(* CODESYS project BE_Framework BA.project

Project tree, tasks and I/O mapping:
  Device : TxB SoftControl, Beijer Electronics Products AB, version 3.5.1.45
    application AREA1
      Symbols
      Struct/
        Sensors/
          data type strSensor1
          data type strSensor2_Regulator
          data type strSensor3_RegOutsideCompensation
          data type strSensor4_FanGuard
          data type strSensor5_FreezeProtection
          data type strSensor6_HeatExchanger_Rot
          data type strSensor7_Humidity
          data type strSensor8_DefrostProtection
          data type strSensor9_CO2
          data type strSensor10_HeatExchanger_Pressure
          data type strSensor11_DifferentialPressure
        Fans/
          data type strFan_Analog
          data type strFan_TwoSpeed
          data type strFan_Onespeed
        Dampers/
          data type strDamper_Digital
          data type strDamper_Analog
        Pumps/
          data type strPumpExercise
          data type strPump
        Valves/
          data type strValveExercise
          data type strValve
        Functions/
          data type strFunction_OutsideCompensation
          data type strFunction_Overtime
          data type strFunction_NightCooling
          data type strFunction_NightHeating
        System/
          data type strSystemTags
          data type strArrayDateTime
          data type strManMode
          data type strSummerTime
        HeatExchangers/
          data type strHeatExchanger_Rot
          data type strHeatExchanger_Cross
        TimeChannels/
          data type strTCH_1StartStop
          data type strTCH_2StartStop
        Units/
          data type strLB
          data type strUC
        IO_Crevis/
          data type strST2792
          data type strST4491
          data type strST1218
          data type strST3708
      System/
        libraries: Standard, * (System); SysTimeRtc, 3.5.1.0 (System); BE Lib BA, 1.1.0.0 (Beijer Electronics)
        task MainTask (cyclic, interval t#20ms, priority 10) calls Sys_SummerPeriod, Sys_CalculateHoliday, Sys_SystemTags, Sys_StartUp, Sys_CommunicationAlarm, LB01_Alarm, LB01_StartConditions, LB01_TimeChannel, LB01_GT81, LB01_GT31_Control, LB01_Cascade_RoomControl, LB01_GT11_RegHeating, LB01_GT11_RegCooling, LB01_GT11, LB01_GT21, LB01_GT41, LB01_P1, LB01_TF1_Analog, LB01_FF1_Analog, LB01_P2, LB01_GP11, LB01_GP21, LB01_GP13, LB01_GP23, LB01_ST11_Digital, LB01_ST21_Digital, LB01_SV61, LB01_SV62, LB01_HeatExchanger_Rot, LB01_GS91, LB01_SequenceHeating, LB01_SequenceCooling, LB01_GT12, LB01_GT13, LB01_GT22, LB01_Function_Dewpoint, LB01_Function_EfficiencyExtractAir, LB01_Function_Overtime, LB01_Function_Preheating, LB01_GM21, LB01_NightCooling, LB01_NightHeating, UCSh1_Alarms, UCSh1_StartConditions, UCSh1_P1, UCSh1_GT1_Control, UCSh1_GT1, UCSh1_GT2, UCSh1_SV1, Sys_Version
        task BusTask (cyclic, interval t#10ms, priority 1) calls AnalogInput, DigitalInput, AnalogOutput, DigitalOutput
        SystemSignals/
          program Sys_SystemTags [CFC]
          program Sys_Version [ST]
        Communication/
          program Sys_CommunicationAlarm [CFC]
          program Sys_StartUp [CFC]
        Functions/
          program Sys_SummerPeriod [CFC]
          program Sys_CalculateHoliday [CFC]
      B001/
        LB01/
          Fan/
            FF1/
              program LB01_FF1_OneSpeed [CFC]
              program LB01_FF1_Analog [CFC]
              program LB01_FF1_TwoSpeed [CFC]
              program LB01_FF1_Analog_ST [ST]
            TF1/
              program LB01_TF1_OneSpeed [CFC]
              program LB01_TF1_TwoSpeed [CFC]
              program LB01_TF1_Analog [CFC]
            FF2/
              program LB01_FF2_Analog_ST [ST]
          Pump/
            P1/
              program LB01_P1 [CFC]
            P2/
              program LB01_P2 [CFC]
            P3/
              program LB01_P3 [CFC]
          Sensor/
            Temperature/
              GT21/
                program LB01_Cascade_ExtractControl [CFC]
                program LB01_GT21 [CFC]
                program LB01_GT21_Control [CFC]
              GT31/
                program LB01_GT31 [CFC]
                program LB01_Cascade_RoomControl [CFC]
                program LB01_GT31_Control [CFC]
              GT41/
                program LB01_GT41 [CFC]
              GT11/
                program LB01_GT11_RegHeating [CFC]
                program LB01_GT11_RegCooling [CFC]
                program LB01_GT11 [CFC]
              GT81/
                program LB01_GT81 [CFC]
              GT12/
                program LB01_GT12 [CFC]
              GT13/
                program LB01_GT13 [CFC]
              GT22/
                program LB01_GT22 [CFC]
              GT91/
                program LB01_GT91 [CFC]
            Pressure/
              GP21/
                program LB01_GP21 [CFC]
              GP11/
                program LB01_GP11 [CFC]
              GP22/
                program LB01_GP22 [CFC]
              GP23/
                program LB01_GP23 [CFC]
              GP13/
                program LB01_GP13 [CFC]
              GP12/
                program LB01_GP12 [CFC]
              GP61/
                program LB01_GP61 [CFC]
              GP91/
                program LB01_GP91 [CFC]
            Flow/
              GF21/
                program LB01_GF21 [CFC]
              GF11/
                program LB01_GF11 [CFC]
            Humidity/
              GM21/
                program LB01_GM21 [CFC]
            Rotationguard/
              program LB01_GS91 [CFC]
          Function/
            program LB01_Function_OutsideCompensation [CFC]
            program LB01_Function_Dewpoint [CFC]
            program LB01_Function_EfficiencyExtractAir [CFC]
            program LB01_Function_EfficiencySupplyAir [CFC]
            program LB01_Function_Overtime [CFC]
            program LB01_Function_Preheating [CFC]
            program LB01_NightCooling [CFC]
            program LB01_NightHeating [CFC]
            program LB01_Function_AirQuality [CFC]
          Sequence/
            program LB01_SequenceHeating [CFC]
            program LB01_SequenceCooling [CFC]
          Valve/
            SV61/
              program LB01_SV61 [CFC]
            SV62/
              program LB01_SV62 [CFC]
            SV91/
              program LB01_SV91 [CFC]
          HeatExchanger/
            program LB01_HeatExchanger_Rot [CFC]
            program LB01_HeatExchanger_Cross [CFC]
          Damper/
            ST11/
              program LB01_ST11_Digital [CFC]
              program LB01_ST11_Analog [CFC]
            ST21/
              program LB01_ST21_Digital [CFC]
              program LB01_ST21_Analog [CFC]
          AirHandlingUnit/
            program LB01_TimeChannel [CFC]
            program LB01_StartConditions [CFC]
            program LB01_Alarm [CFC]
        global variables GVL_B001
        global variables B001
        UC/
          Sh1/
            Pump/
              program UCSh1_P1 [CFC]
            Valve/
              program UCSh1_SV1 [CFC]
            Sensor/
              GT1/
                program UCSh1_GT1_Control [CFC]
                program UCSh1_GT1 [CFC]
              GT2/
                program UCSh1_GT2 [CFC]
            Alarms/
              program UCSh1_Alarms [CFC]
            UcUnit/
              program UCSh1_StartConditions [CFC]
      IO/
        Input/
          program DigitalInput [CFC]
          program AnalogInput [CFC]
        Output/
          program DigitalOutput [CFC]
          program AnalogOutput [CFC]
      FB/
        function block FB_SystemSignals [ST]
      Testing Center/
        program Test [ST]
    Ethernet : Ethernet, 3S - Smart Software Solutions GmbH, version 3.4.2.0
      Modbus_TCP_Master : Modbus TCP Master, 3S - Smart Software Solutions GmbH, version 3.5.1.0
          settings: AutoReconnect = TRUE
        Modbus_TCP_Slave : Modbus TCP Slave, 3S - Smart Software Solutions GmbH, version 3.5.1.0
            settings: 16#2011 (=8209).Function Code = 16; 16#2011 (=8209).Write Offset = 8209; 16#2011 (=8209).Write Length = 1; 16#2011 (=8209).Init Value = 3; Unit-ID = 1; IPAddress = [192, 168, 1, 11]; Channel 0.Function Code = 23; Channel 0.Read Offset = 16#0000; Channel 0.Read Length = 12; Channel 0.Write Offset = 16#0800; Channel 0.Write Length = 2; Channel 0.Cycle Time = 100
            input  AREA1.Nod1_Slot1.ST3708_AI1 : WORD  // Channel 0.Channel 0[0]
            input  AREA1.Nod1_Slot1.ST3708_AI2 : WORD  // Channel 0.Channel 0[1]
            input  AREA1.Nod1_Slot1.ST3708_AI3 : WORD  // Channel 0.Channel 0[2]
            input  AREA1.Nod1_Slot1.ST3708_AI4 : WORD  // Channel 0.Channel 0[3]
            input  AREA1.Nod1_Slot1.ST3708_AI5 : WORD  // Channel 0.Channel 0[4]
            input  AREA1.Nod1_Slot1.ST3708_AI6 : WORD  // Channel 0.Channel 0[5]
            input  AREA1.Nod1_Slot1.ST3708_AI7 : WORD  // Channel 0.Channel 0[6]
            input  AREA1.Nod1_Slot1.ST3708_AI8 : WORD  // Channel 0.Channel 0[7]
            input  AREA1.Nod1_Slot2.ST4491_Switch1DI1 : BOOL  // Channel 0.Channel 0[8].Bit0
            input  AREA1.Nod1_Slot2.ST4491_Switch2AI1 : WORD  // Channel 0.Channel 0[9]
            input  AREA1.Nod1_Slot3.ST1218_DI1 : BOOL  // Channel 0.Channel 0[10].Bit0
            input  AREA1.Nod1_Slot3.ST1218_DI2 : BOOL  // Channel 0.Channel 0[10].Bit1
            input  AREA1.Nod1_Slot3.ST1218_DI3 : BOOL  // Channel 0.Channel 0[10].Bit2
            input  AREA1.Nod1_Slot3.ST1218_DI4 : BOOL  // Channel 0.Channel 0[10].Bit3
            input  AREA1.Nod1_Slot3.ST1218_DI5 : BOOL  // Channel 0.Channel 0[10].Bit4
            input  AREA1.Nod1_Slot3.ST1218_DI6 : BOOL  // Channel 0.Channel 0[10].Bit5
            input  AREA1.Nod1_Slot3.ST1218_DI7 : BOOL  // Channel 0.Channel 0[10].Bit6
            input  AREA1.Nod1_Slot3.ST1218_DI8 : BOOL  // Channel 0.Channel 0[10].Bit7
            input  AREA1.Nod1_Slot4.ST2792_Switch1DI1 : BOOL  // Channel 0.Channel 0[10].Bit8
            input  AREA1.Nod1_Slot4.ST2792_Switch2DI1 : BOOL  // Channel 0.Channel 0[10].Bit9
            input  AREA1.Nod1_Slot4.ST2792_Switch1DI2 : BOOL  // Channel 0.Channel 0[11].Bit0
            input  AREA1.Nod1_Slot4.ST2792_Switch2DI2 : BOOL  // Channel 0.Channel 0[11].Bit1
            output AREA1.Nod1_Slot2.ST4491_AO1 : WORD  // Channel 0.Channel 0[0]
            output AREA1.Nod1_Slot4.ST2792_DO1 : BOOL  // Channel 0.Channel 0[1].Bit0
            output AREA1.Nod1_Slot4.ST2792_DO2 : BOOL  // Channel 0.Channel 0[1].Bit1
            unmapped channels: Channel 0, Channel 0
  libraries: AC_ModuleBase, * (3S - Smart Software Solutions GmbH); AC_DeviceDiagnosis, 3.5.4.0 (3S - Smart Software Solutions GmbH); AC_Persistence, 3.5.4.0 (3S - Smart Software Solutions GmbH)
*)

// Device/AREA1/Struct/Fans/strFan_Analog
TYPE strFan_Analog :
STRUCT
	OP:REAL;									//Output value																@0;100;0;100;%; ### EU;T
	AUT:INT;									//0=Auto, 1=Off, 2=On														@
	AL:BOOL;									//General alarm
	AL01:BOOL;									//Feedback error																@AL01
	AL02:BOOL;									//Thermal relay triggered													@AL01
	V:BOOL;										// On/Open																	@
	CMD:BOOL;									//Commanded start															@
	SP1:DINT;									//Start delay																	@0;3200;0;3200;s; #### EU
	SP2:DINT;									//Thermal Relay alarm delay											@0;3200;0;3200;s; #### EU
	SP3:DINT;									//Fan guard alarm delay													@0;3200;0;3200;s; #### EU
	SP4:DINT;									//Feedback alarm delay													@0;3200;0;3200;s; #### EU
	OPM:REAL;									//Manual output																@0;100;0;100;%; ###.# EU
	ACK:BOOL;									//Acknowledge alarm

	//Operating Time
	PV1:DINT;									//Total operating hours													@0;9999999;0;9999999;tim; ####### EU
	PV2:INT;										//Total operating minutes 												@0;59;0;59;min; ## EU	
	PV3:DINT;									//Total number of starts since reset									@0;9999999;0;9999999;st; ####### EU
	RST:BOOL;									//Resetting the operation time and number of starts			@	
	
	//Hardware switches
	ST2792_M:BOOL;							//Manual operating mode from hardware
	ST2792_MCMD:BOOL;					//Manual commanded starting from hardware
	ST4491_M:BOOL;							//Manual mode for analog value from hardware
	ST4491_OPM:REAL;						//Manual output value from hardware
	
	//Not used in Scada
	Symbol:INT;								//Symbol Value (0-3)
	Symbol_M:INT;							//Symbol in manual mode
	Operating:BOOL;							//Objects in operation
	StatusOff:BOOL;							//Stopped in manual mode
	StatusOn:BOOL;							//Started in manual mode
	SumAlarm:BOOL;							//General alarm
	RunIndication:BOOL;					//Operating indicator
	ManualStart:BOOL;						//Manual start command
	EnFeedbackError:BOOL;				//Activate feedback alarm
	FeedbackError:BOOL;					//Feedback error
	EnThermalError:BOOL;					//Activate Thermal Relay alarm
	ThermalError:BOOL;						//Thermal relay fault
	EnFanGuardError:BOOL;				//Activate Fan Guard error
	FanGuardError:BOOL;					//Fan Guard error
	ThermoRelay1:BOOL;					//Thermal Relay ok, halfspeed
END_STRUCT
END_TYPE

// Device/AREA1/Struct/Sensors/strSensor1
TYPE strSensor1 :
STRUCT
	PV:REAL;									//Process value																@0;4095;0;100;°C; ###.# EU;T2
	AD:DINT;									//Alarm Delay																@0;65535;-1000;1500;min; ### EU;;R1
	AL:BOOL;									//General alarm	
	FAULT:BOOL;									//Sensor error																@AL02
	LAL:BOOL;									//Low alarm																	@AL02
	HAL:BOOL;									//High alarm																@AL02
	ALL:REAL;									//Low alarm level															@-99;100;-99;100;°C; ###.# EU;T1;R2
	AHL:REAL;									//High alarm level															@-99;100;-99;100;°C; ###.# EU
	ACK:BOOL;									//Acknowledge alarm
	
	//Not used in Scada
	En:BOOL;									//Enable controll
	Symbol:INT;									//Symbol Value (0-3)
END_STRUCT
END_TYPE

// Device/AREA1/Struct/Sensors/strSensor2_Regulator
TYPE strSensor2_Regulator :
STRUCT
	PV:REAL;									//Process value																@-99;100;-99;100;°C; ###.# EU;T
	SP:REAL;									//Setpoint																		@-99;100;-99;100;°C; ###.# EU;T
	CSP:REAL;									//Calculated setpoint														@-99;100;-99;100;°C; ###.# EU;T
	CSP1:REAL;									//Calculated low alarm level												@-99;100;-99;100;°C; ###.# EU;T
	CSP2:REAL;									//Calculated high alarm level											@-99;100;-99;100;°C; ###.# EU;T
	AD:DINT;									//Alarm Delay																@0;999;0;999;min; ### EU
	AL:BOOL;									//General alarm	
	FAULT:BOOL;								//Sensor error																	@AL02
	ALL:REAL;									//Low alarm level															@-99;100;-99;100;°C; ###.# EU
	AHL:REAL;									//High alarm level															@-99;100;-99;100;°C; ###.# EU
	ADL:REAL;									//Deviation ±																	@0;100;0;100;°C; ###.# EU
	P:REAL;										//Proportional constant													@0;9999;0;9999;; ####.# EU
	I:REAL;										//Integral																		@0;9999;0;9999;s; ####.# EU
	D:REAL;										//Derivation																	@0;9999;0;9999;s; ####.# EU
	SI:REAL;										//Sample time
	DB:REAL;									//Dead band
	MAX1:REAL;								//Maximum output from regulator									@0;100;0;100;%; ### EU
	MIN1:REAL;								//Minimum output from regulator										@0;100;0;100;%; ### EU
	M:BOOL;									//Manual mode
	OPM:REAL;									//Manual output																@0;100;0;100;%; ###.# EU
	OP:REAL;									//Output value (från regulatorn)										@0;100;0;100;%; ### EU
	LAL:BOOL;									//Low temperature															@AL02
	HAL:BOOL;									//High temperature															@AL02
	SP1:REAL;									//Min input value (cascade control)									@-99;100;-99;100;°C; ###.# EU
	SP2:REAL;									//Max input value (cascade control)									@-99;100;-99;100;°C; ###.# EU
	SP3:REAL;									//Dead zone, regulating heat to cold									@0;100;0;100;°C; ###.# EU
	ACK:BOOL;									//Acknowledge alarm

	//Not used in Scada
	En:BOOL;									//Enable controll
	Symbol:INT;								//Symbol Value (0-3)
	PID_En:BOOL;								//Enable PID control
	SavedData:ARRAY [0..15] OF REAL;	//Saved data for the object		
END_STRUCT
END_TYPE

// Device/AREA1/Struct/Sensors/strSensor3_RegOutsideCompensation
TYPE strSensor3_RegOutsideCompensation:
STRUCT
	PV:REAL;									//Process value																@-99;100;-99;100;°C; ###.# EU;T
	SP:REAL;									//Setpoint																		@-99;100;-99;100;°C; ###.# EU;T
	CSP:REAL;									//Calculated setpoint														@-99;100;-99;100;°C; ###.# EU;T
	CSP1:REAL;									//Calculated low alarm level												@-99;100;-99;100;°C; ###.# EU;T
	CSP2:REAL;									//Calculated high alarm level											@-99;100;-99;100;°C; ###.# EU;T
	AD:DINT;									//Alarm Delay																@0;999;0;999;min; ### EU
	AL:BOOL;									//General alarm	
	FAULT:BOOL;								//Sensor error																	@AL02
	ALL:REAL;									//Low alarm level															@-99;100;-99;100;°C; ###.# EU
	AHL:REAL;									//High alarm level															@-99;100;-99;100;°C; ###.# EU
	ADL:REAL;									//Deviation ±																	@0;100;0;100;°C; ###.# EU
	P:REAL;										//Proportional constant													@0;9999;0;9999;; ####.# EU
	I:REAL;										//Integral																		@0;9999;0;9999;s; ####.# EU
	D:REAL;										//Derivation																	@0;9999;0;9999;s; ####.# EU
	SI:REAL;										//Sample time
	DB:REAL;									//Dead band
	MAX1:REAL;								//Maximum output from regulator									@0;100;0;100;%; ### EU
	MIN1:REAL;								//Minimum output from regulator										@0;100;0;100;%; ### EU
	M:BOOL;									//Manual mode
	OPM:REAL;									//Manual output																@0;100;0;100;%; ###.# EU
	OP:REAL;									//Output value (från regulatorn)										@0;100;0;100;%; ### EU
	LAL:BOOL;									//Low temperature															@AL02
	HAL:BOOL;									//High temperature															@AL02
	SP1:REAL;									//Min input value (cascade control)									@-99;100;-99;100;°C; ###.# EU
	SP2:REAL;									//Max input value (cascade control)									@-99;100;-99;100;°C; ###.# EU
	SP3:REAL;									//Dead zone, regulating heat to cold									@0;100;0;100;°C; ###.# EU
	ACK:BOOL;									//Acknowledge alarm

	CSP3:REAL;									//Outcompensation setpoint												@-99;100;-99;100;°C; ###.# EU
	Y1:REAL;									//Break point Y1 for output signal.									@-99;100;-99;100;°C; ###.# EU
	Y2:REAL;									//Break point Y2 for output signal.									@-99;100;-99;100;°C; ###.# EU
	Y3:REAL;									//Break point Y3 for output signal.									@-99;100;-99;100;°C; ###.# EU
	Y4:REAL;									//Break point Y4 for output signal.									@-99;100;-99;100;°C; ###.# EU
	Y5:REAL;									//Break point Y5 for output signal.									@-99;100;-99;100;°C; ###.# EU
	Y6:REAL;									//Break point Y6 for output signal.									@-99;100;-99;100;°C; ###.# EU
	Y7:REAL;									//Break point Y7 for output signal.									@-99;100;-99;100;°C; ###.# EU
	Y8:REAL;									//Break point Y8 for output signal.									@-99;100;-99;100;°C; ###.# EU
	X1:REAL;									//Break point X1 for input signal.										@-99;100;-99;100;°C; ###.# EU
	X2:REAL;									//Break point X2 for input signal.										@-99;100;-99;100;°C; ###.# EU
	X3:REAL;									//Break point X3 for input signal.										@-99;100;-99;100;°C; ###.# EU
	X4:REAL;									//Break point X4 for input signal.										@-99;100;-99;100;°C; ###.# EU
	X5:REAL;									//Break point X5 for input signal.										@-99;100;-99;100;°C; ###.# EU
	X6:REAL;									//Break point X6 for input signal.										@-99;100;-99;100;°C; ###.# EU
	X7:REAL;									//Break point X7 for input signal.										@-99;100;-99;100;°C; ###.# EU
	X8:REAL;									//Break point X8 for input signal.										@-99;100;-99;100;°C; ###.# EU

	//Not used in Scada
	Symbol:INT;								//Symbol Value (0-3)
	En:BOOL;									//Enable function
	PID_En:BOOL;								//Enable PID control
	SavedData:ARRAY [0..15] OF REAL;	//Saved data for the object	
END_STRUCT
END_TYPE

// Device/AREA1/Struct/Functions/strFunction_OutsideCompensation
TYPE strFunction_OutsideCompensation :
STRUCT
	CSP3:REAL;									//Setpoint Outdoor Compensation.										@-99;100;-99;100;°C; ###.# EU
	Y1:REAL;									//Break point Y1 for output signal.									@-99;100;-99;100;°C; ###.# EU
	Y2:REAL;									//Break point Y2 for output signal.									@-99;100;-99;100;°C; ###.# EU
	Y3:REAL;									//Break point Y3 for output signal.									@-99;100;-99;100;°C; ###.# EU
	Y4:REAL;									//Break point Y4 for output signal.									@-99;100;-99;100;°C; ###.# EU
	Y5:REAL;									//Break point Y5 for output signal.									@-99;100;-99;100;°C; ###.# EU
	Y6:REAL;									//Break point Y6 for output signal.									@-99;100;-99;100;°C; ###.# EU
	Y7:REAL;									//Break point Y7 for output signal.									@-99;100;-99;100;°C; ###.# EU
	Y8:REAL;									//Break point Y8 for output signal.									@-99;100;-99;100;°C; ###.# EU
	X1:REAL;									//Break point X1 for input signal.										@-99;100;-99;100;°C; ###.# EU
	X2:REAL;									//Break point X2 for input signal.										@-99;100;-99;100;°C; ###.# EU
	X3:REAL;									//Break point X3 for input signal.										@-99;100;-99;100;°C; ###.# EU
	X4:REAL;									//Break point X4 for input signal.										@-99;100;-99;100;°C; ###.# EU
	X5:REAL;									//Break point X5 for input signal.										@-99;100;-99;100;°C; ###.# EU
	X6:REAL;									//Break point X6 for input signal.										@-99;100;-99;100;°C; ###.# EU
	X7:REAL;									//Break point X7 for input signal.										@-99;100;-99;100;°C; ###.# EU
	X8:REAL;									//Break point X8 for input signal.										@-99;100;-99;100;°C; ###.# EU
	
	//Not used in Scada
	En:BOOL;									//Enable function
END_STRUCT
END_TYPE

// Device/AREA1/Struct/Sensors/strSensor4_FanGuard
TYPE strSensor4_FanGuard :
STRUCT
	V:BOOL;										//Status
	AD:DINT;									//Alarm Delay																@0;999;0;999;min; ### EU
	AL:BOOL;									//General alarm	
	AL01:BOOL;									//Filter guard alarm														@AL01
	ACK:BOOL;									//Acknowledge alarm

	//Not used in Scada
	Symbol:INT;								//Symbol Value (0-3)
END_STRUCT
END_TYPE

// Device/AREA1/Struct/Fans/strFan_TwoSpeed
TYPE strFan_TwoSpeed:
STRUCT
	M:BOOL;									//Manual mode																@
	AL:BOOL;									//General alarm
	AL01:BOOL;									//Feedback error																@AL01
	AL02:BOOL;									//Thermal relay triggered													@AL01
	SP1:DINT;									//Start delay																	@0;3200;0;3200;s; #### EU
	SP2:DINT;									//Thermal Relay alarm delay											@0;3200;0;3200;s; #### EU
	SP3:DINT;									//Fan guard alarm delay													@0;3200;0;3200;s; #### EU
	SP4:DINT;									//Feedback alarm delay													@0;3200;0;3200;s; #### EU
	ACK:BOOL;									//Acknowledge alarm
	MCMD1:BOOL;								//Manually commanded full speed										@
	MCMD2:BOOL;								//Manually commanded half speed									@
	AL03:BOOL;									//Half speed feedback alarm									  			@AL01
	AL04:BOOL;									//Half speed thermal relay triggered									@AL01
	AL05:BOOL;									//Full speed feedback alarm 											@AL01
	AL06:BOOL;									//Full speed thermal relay alarm										@AL01
	V1:BOOL;									//Feedback full speed														@
	V2:BOOL;									//Feedback half speed 														@
	CMD1:BOOL;								//Commanded start full speed											@
	CMD2:BOOL;								//Commanded start half speed 											@
	SP5:INT;										//Delay from half speed to full speed								@0;3200;0;3200;s; #### EU
	SP6:INT;										//Delay from full speed to half speed								@0;3200;0;3200;s; #### EU

	//Operating Time
	PV1:DINT;									//Total operating hours													@0;9999999;0;9999999;tim; ####### EU
	PV2:INT;										//Total operating minutes 												@0;59;0;59;min; ## EU	
	PV3:DINT;									//Total number of starts since reset									@0;9999999;0;9999999;st; ####### EU
	RST:BOOL;									//Resetting the operation time and number of starts			@	

	//Hardware switches
	ST2792_M:BOOL;							//Manual operating mode from hardware
	ST2792_MCMD:BOOL;					//Manual commanded starting from hardware
	ST4491_M:BOOL;							//Manual mode for analog value from hardware
	ST4491_OPM:REAL;						//Manual output value from hardware
	
	//Not used in Scada
	Symbol:INT;								//Symbol Value (0-3)
	Symbol_M:INT;							//Symbol in manual mode
	Operating:BOOL;							//Objects in operation
	StatusOff:BOOL;							//Stopped in manual mode
	StatusOn:BOOL;							//Started in manual mode
	SumAlarm:BOOL;							//General alarm
	RunIndication:BOOL;					//Operating indicator
	ManualStart:BOOL;						//Manual start command-
	EnFeedbackError:BOOL;				//Activate feedback alarm
	FeedbackError:BOOL;					//Feedback error
	EnThermalError:BOOL;					//Activate Thermal Relay alarm
	ThermalError:BOOL;						//Thermal relay fault
	EnFanGuardError:BOOL;				//Activate Fan Guard error
	FanGuardError:BOOL;					//Fan Guard error
	FS_StatusOff:BOOL;						//Helfart stoppad i manuellt läge
	FS_StatusOn:BOOL;						//Helfart startad i manuellt läge
	HS_StatusOff:BOOL;						//Halvfart stoppad i manuellt läge
	HS_StatusOn:BOOL;						//Halvfart startad i manuellt läge
	StartTwoSpeed:BOOL;					//Kommenderad helfart
	ThermoRelay1:BOOL;					//Thermal Relay ok, halfspeed
	ThermoRelay2:BOOL;					//Termorelä ok helfart
	FeedbackError1:BOOL;					//Feedback error halvfart
	FeedbackError2:BOOL;					//Feedback error helfart
	ThermalError1:BOOL;					//Thermal relay fault halvfart
	ThermalError2:BOOL;					//Thermal relay fault helfart
END_STRUCT
END_TYPE

// Device/AREA1/Struct/Valves/strValveExercise
TYPE strValveExercise :
STRUCT
	AUT:INT;									//0=Auto, 1=Off, 2=On														@
	OP:REAL;									//Output value																@0;100;0;100;%; ### EU;T
	OPM:REAL;									//Manual output																@0;100;0;100;%; ###.# EU
	V:BOOL;										// On/Open																	@
	SP1:INT;										//Number of days before exercise										@0;999;0;999;dag; ### EU
	SP2:INT;										//Number of hours before exercise									@0;23;0;23;tim; ## EU
	
	//Excercise
	PV1:INT;										//Days before exercise														@0;999;0;999;dag; ### EU
	PV2:INT;										//Hours before exercise													@0;23;0;23;tim; ## EU
	PV3:INT;										//Minutes before exercise 												@0;59;0;59;min; ## EU	
	SP3:INT;										//Starting day exercise														@0;6;0;6;dag; # EU
	SP4:INT;										//Starting time exercise													@0;23;0;23;tim; ## EU
	SP5:INT;										//Starting time exercise 													@0;59;0;59;min; ## EU
	SP6:INT;										//Exercise time 																@0;999;0;999;min; ### EU
	V01:BOOL;									//Status exercise																@
	
	//Hardware switches
	ST2792_M:BOOL;							//Manual operating mode from hardware
	ST2792_MCMD:BOOL;					//Manual commanded starting from hardware
	ST4491_M:BOOL;							//Manual mode for analog value from hardware
	ST4491_OPM:REAL;						//Manual output value from hardware
	
	//Not used in Scada
	Frost_V:BOOL;								//Antifreeze activated
	Frost_En:BOOL;							//Enable antifreeze
	Symbol_M:INT;							//Symbol in manual mode
	Seq_Output:REAL;						//Control range of valve
	Ex_En:BOOL;								//Enable exercise
	Ex_En_Day:BOOL;							//Enable specific day
	Ex_En_Time:BOOL;						//Enable specific time	
	Ex_SecOff:DINT;							//Enumeration of seconds when the object is not in operation
	Ex_SavedData:ARRAY [0..3] OF INT;//Saved data for the object	
END_STRUCT
END_TYPE

// Device/AREA1/Struct/Dampers/strDamper_Digital
TYPE strDamper_Digital :
STRUCT
	CMD:BOOL;									//Command open															@
	AUT:INT;									//0=Auto, 1=Off, 2=On														@
	V:BOOL;										// On/Open																	@
	
	//Hardware switches
	ST2792_M:BOOL;							//Manual operating mode from hardware
	ST2792_MCMD:BOOL;					//Manual commanded starting from hardware
	ST4491_M:BOOL;							//Manual mode for analog value from hardware
	ST4491_OPM:REAL;						//Manual output value from hardware
	
	//Not used in Scada
	Symbol_M:INT;							//Symbol in manual mode
	StatusOff:BOOL;							//Stopped in manual mode
	StatusOn:BOOL;							//Started in manual mode
END_STRUCT
END_TYPE

// Device/AREA1/Struct/System/strSystemTags
TYPE strSystemTags :
STRUCT
	xAlwaysFalse:BOOL;										//Signal will always be FALSE
	xAlwaysTrue:BOOL;										//Signal will always be TRUE

	xOnFirstScan:BOOL;										//ON at the first PLC scan
	xOffFirstScan:BOOL;										//OFF at the first scan
	
	xFlash2s:BOOL;											//ON for 1000ms / OFF for 1000ms
	xFlash1s:BOOL;											//ON for 500ms / OFFfor 500ms
	xFlash100ms:BOOL;										//ON for 50ms / OFF for 50ms
	
	xPulseMinute:BOOL;									//ON for one scan each minute
	xPulse1s:BOOL;											//ON for one scan each second
	xPulse100ms:BOOL;										//ON for one scan each 100ms
	
	xCurrentTimeAndDate:RTS_SYSTIMEDATE;		//Date and Time struct

	xNewDayPulse:BOOL;									//New day pulse (will trig for one scan 23:59 each night)
END_STRUCT
END_TYPE

// Device/AREA1/Struct/System/strArrayDateTime
TYPE strArrayDateTime :
STRUCT
	Year:UINT;									//Year
	Month:UINT;								//Month
	Day:UINT;									//Day
	Hour:UINT;									//Hour
	Minute:UINT;								//Minute
	Second:UINT;								//Second
	DayOfWeek:UINT;						//Day of week
END_STRUCT
END_TYPE

// Device/AREA1/Struct/Units/strLB
TYPE strLB :
STRUCT
	//Sensors
	GT31:strSensor2_Regulator;									//Room temperature sensor
	GT11:strSensor2_Regulator;									//Supply air temperature sensor
	GT11_Cool:strSensor2_Regulator;							//Supply air temperature sensor
	GT12:strSensor1;													//Intake air temperature sensor
	GT13:strSensor1;													//Supply air temperature sensor after heatexchanger
	GT21:strSensor1;													//Extract air temperature sensor
	GT22:strSensor1;													//Exhaust air temperature sensor
	GT41:strSensor1;													//Outdoor temperature sensor
	GT81:strSensor5_FreezeProtection;						//Freeze sensor
	GP11:strSensor2_Regulator;									//Supply air pressure sensor
	GP13:strSensor4_FanGuard;									//Differential pressure TF1
	GP21:strSensor2_Regulator;									//Extract air pressure sensor
	GP23:strSensor4_FanGuard;									//Differential pressure FF1
	GS91:strSensor6_HeatExchanger_Rot;						//Rotationguard
	GM21:strSensor7_Humidity;									//Humidity sensor
	
	//Fans
	TF1:strFan_Analog;												//Supply air fan
	FF1:strFan_Analog;												//Exhaust air fan
	
	//Pumps
	P1:strPumpExercise;											//Heat pump
	P2:strPumpExercise;											//Cooling pump
	
	//Valves
	SV61:strValve;														//Heat valve
	SV62:strValve;														//Cooling valve
	
	//Dampers
	ST11:strDamper_Digital;										//Intake damper
	ST21:strDamper_Digital;										//Exhaust damper
	
	//HeatExchanger
	VVX:strHeatExchanger_Rot;									//Heat exchanger
	
	//TimeChannels
	TCH01:strTCH_1StartStop;										//Time channel

	//Functions
	Overtime:strFunction_Overtime;							//Function Overtime
	NC:strFunction_NightCooling;								//Function Night cooling
	NH:strFunction_NightHeating;								//Function Night heating
	
	//Misc signals
	ManMode:strManMode;										//Alarm when one or more objects are too long in manual
	A_Alarm:BOOL;													//General alarms A-larm
	GeneralStart:BOOL;												//Air unit started						@
	Heat_RegOutput:REAL;										//Scaled output value from the controller
	AlarmStatusReg:INT;												//Status for alarm symbol
	FireAlarm:BOOL;													//Input fire alarm
	SWITCH:INT;														//Switch for the air unit		0=Off, 1=Manual, 2=Auto
	System_Nod1_AL:BOOL;										//Communication alarm
	System_Nod1_Count:INT;										//Count node alarm
	System_Nod_RST:BOOL;										//Reset of communication alarm
END_STRUCT
END_TYPE

// Device/AREA1/Struct/Sensors/strSensor5_FreezeProtection
TYPE strSensor5_FreezeProtection :
STRUCT
	PV:REAL;									//Process value																@-99;100;-99;100;°C; ###.# EU;T
	AD:DINT;									//Alarm Delay																@0;999;0;999;min; ### EU
	AL:BOOL;									//General alarm	
	FAULT:BOOL;								//Sensor error																	@AL02
	ALL:REAL;									//Low alarm level															@-99;100;-99;100;°C; ###.# EU
	AHL:REAL;									//High alarm level															@-99;100;-99;100;°C; ###.# EU
	AL01:BOOL;									//Freeze protection activated											@AL01
	HAL:BOOL;									//High temperature															@AL02
	LAL:BOOL;									//Low temperature															@AL02
	SP:REAL;									//Keeping warm when the aggregate is off 							@-99;100;-99;100;°C; ###.# EU
	SP2:REAL;									//Minimum limit when operating										@-99;100;-99;100;°C; ###.# EU
	SP1:REAL;									//Freeze Protection															@-99;100;-99;100;°C; ###.# EU
	OP:REAL;									//Output value																@0;100;0;100;%; ### EU
	ACK:BOOL;									//Acknowledge alarm

	//Not used in Scada
	Symbol:INT;								//Symbol Value (0-3)
	FreezeProtect:BOOL;					//Freeze protection activated
END_STRUCT
END_TYPE

// Device/AREA1/Struct/HeatExchangers/strHeatExchanger_Rot
TYPE strHeatExchanger_Rot :
STRUCT
	AUT:INT;									//0=Auto, 1=Off, 2=On														@
	OP:REAL;									//Output value																@0;100;0;100;%; ### EU;T
	OPM:REAL;									//Manual output																@0;100;0;100;%; ###.# EU
	V:BOOL;										// On/Open																	@
	AL:BOOL;									//General alarm
	ACK:BOOL;									//Acknowledge alarm

	//Verkningsgradsberäkning
	PV1:REAL;									//Calculated efficiency													@0;100;0;100;%; ### EU;T
	AD:DINT;									//Efficiency, Alarm delay													@0;9999;0;9999;min; #### EU
	ALL:REAL;									//Efficiency, Alarm level 													@0;100;0;100;%; ###.# EU
	LAL:BOOL;									//Low efficiency																@AL02
	AL01:BOOL;									//Efficiency alarm
	
	//Kylåtervinning
	V01:BOOL;									//Cooling recovery activated												@
	SP3:REAL;									//Temperature difference for cooling recovery					@0;100;0;100;°C; ###.# EU
	
	//Preheating
	OP01:REAL;								//Calculated preheating value											@-99;100;-99;100;min; ###.# EU
	SP4:DINT;									//Preheating time															@0;9999;0;9999;min; #### EU
	SP5:REAL;									//The lowest outdoor temperature for preheating				@-99;100;-99;100;min; ###.# EU
	SP6:REAL;									//The highest outdoor temperature for preheating				@-99;100;-99;100;min; ###.# EU
	V02:BOOL;									//Preheating activated														@
	
	//Hardware switches
	ST2792_M:BOOL;							//Manual operating mode from hardware
	ST2792_MCMD:BOOL;					//Manual commanded starting from hardware
	ST4491_M:BOOL;							//Manual mode for analog value from hardware
	ST4491_OPM:REAL;						//Manual output value from hardware
	
	//Not used in Scada
	Symbol:INT;								//Symbol Value (0-3)
	Symbol_M:INT;							//Symbol in manual mode
	Seq_Heating:REAL;						//Control range of heat recovery
	Seq_Cooling:REAL;						//Control range for cooling recovery
	Eff_En:BOOL;								//Enable function
	CoolingRecycling_En:BOOL;			//Enable function
	Preheating_En:BOOL;					//Enable function
END_STRUCT
END_TYPE

// Device/AREA1/Struct/Sensors/strSensor6_HeatExchanger_Rot
TYPE strSensor6_HeatExchanger_Rot :
STRUCT
	AL:BOOL;									//General alarm	
	AL01:BOOL;									//Rotation control triggered												@AL02
	InputAlarm:BOOL;						//Alarm signal
	ACK:BOOL;									//Acknowledge alarm
	AD:DINT;									//Alarm Delay																@0;999;0;999;min; ### EU

	//Not used in Scada
	Symbol:INT;								//Symbol Value (0-3)
END_STRUCT
END_TYPE

// Device/AREA1/Struct/TimeChannels/strTCH_1StartStop
TYPE strTCH_1StartStop :
STRUCT
	En:BOOL;									//Enable Scheduler with a start and stop per day
	Arr:ARRAY [0..17] OF INT;
	CT1:INT;										//Monday: Start time 1													@0000;2359;0000;2359;hhmm; ####
	CT2:INT;										//Tuesday: Start time 1													@0000;2359;0000;2359;hhmm; ####
	CT3:INT;										//Wednesday: Start time 1												@0000;2359;0000;2359;hhmm; ####
	CT4:INT;										//Thursday: Start time 1													@0000;2359;0000;2359;hhmm; ####
	CT5:INT;										//Friday: Start time 1														@0000;2359;0000;2359;hhmm; ####
	CT6:INT;										//Saturday: Start time 1													@0000;2359;0000;2359;hhmm; ####
	CT7:INT;										//Sunday: Start time 1														@0000;2359;0000;2359;hhmm; ####
	CT8:INT;										//Eve: Start time 1															@0000;2359;0000;2359;hhmm; ####
	CT9:INT;										//Holiday: Start time 1													@0000;2359;0000;2359;hhmm; ####
	CF1:INT;										//Monday: Stop time 1														@0000;2359;0000;2359;hhmm; ####
	CF2:INT;										//Tuesday: Stop time 1													@0000;2359;0000;2359;hhmm; ####
	CF3:INT;										//Wednesday: Stop time 1												@0000;2359;0000;2359;hhmm; ####
	CF4:INT;										//Thursday: Stop time 1													@0000;2359;0000;2359;hhmm; ####
	CF5:INT;										//Friday: Stop time 1														@0000;2359;0000;2359;hhmm; ####
	CF6:INT;										//Saturday: Stop time 1													@0000;2359;0000;2359;hhmm; ####
	CF7:INT;										//Sunday: Stop time 1														@0000;2359;0000;2359;hhmm; ####
	CF8:INT;										//Eve: Stop time 1															@0000;2359;0000;2359;hhmm; ####
	CF9:INT;										//Holiday: Stop time 1														@0000;2359;0000;2359;hhmm; ####
	V:BOOL;										//Time channel is active
END_STRUCT
END_TYPE

// Device/AREA1/Struct/TimeChannels/strTCH_2StartStop
TYPE strTCH_2StartStop :
STRUCT
	En:BOOL;									//Aktivera Tidkanal med två start och stopp per dag
	Arr:ARRAY [0..35] OF INT;
	CT1:INT;										//Monday: Start time 1													@0000;2359;0000;2359;hhmm; ####
	CT2:INT;										//Tuesday: Start time 1													@0000;2359;0000;2359;hhmm; ####
	CT3:INT;										//Wednesday: Start time 1												@0000;2359;0000;2359;hhmm; ####
	CT4:INT;										//Thursday: Start time 1													@0000;2359;0000;2359;hhmm; ####
	CT5:INT;										//Friday: Start time 1														@0000;2359;0000;2359;hhmm; ####
	CT6:INT;										//Saturday: Start time 1													@0000;2359;0000;2359;hhmm; ####
	CT7:INT;										//Sunday: Start time 1														@0000;2359;0000;2359;hhmm; ####
	CT8:INT;										//Eve: Start time 1															@0000;2359;0000;2359;hhmm; ####
	CT9:INT;										//Holiday: Start time 1													@0000;2359;0000;2359;hhmm; ####
	CT11:INT;									//Monday: Start time 2													@0000;2359;0000;2359;hhmm; ####
	CT12:INT;									//Tuesday: Start time 2													@0000;2359;0000;2359;hhmm; ####
	CT13:INT;									//Wednesday: Start time 2												@0000;2359;0000;2359;hhmm; ####
	CT14:INT;									//Thursday: Start time 2													@0000;2359;0000;2359;hhmm; ####
	CT15:INT;									//Friday: Start time 2														@0000;2359;0000;2359;hhmm; ####
	CT16:INT;									//Saturday: Start time 2													@0000;2359;0000;2359;hhmm; ####
	CT17:INT;									//Sunday: Start time 2														@0000;2359;0000;2359;hhmm; ####
	CT18:INT;									//Eve: Start time 2															@0000;2359;0000;2359;hhmm; ####
	CT19:INT;									//Holiday: Start time 2													@0000;2359;0000;2359;hhmm; ####
	CF1:INT;										//Monday: Stop time 1														@0000;2359;0000;2359;hhmm; ####
	CF2:INT;										//Tuesday: Stop time 1													@0000;2359;0000;2359;hhmm; ####
	CF3:INT;										//Wednesday: Stop time 1												@0000;2359;0000;2359;hhmm; ####
	CF4:INT;										//Thursday: Stop time 1													@0000;2359;0000;2359;hhmm; ####
	CF5:INT;										//Friday: Stop time 1														@0000;2359;0000;2359;hhmm; ####
	CF6:INT;										//Saturday: Stop time 1													@0000;2359;0000;2359;hhmm; ####
	CF7:INT;										//Sunday: Stop time 1														@0000;2359;0000;2359;hhmm; ####
	CF8:INT;										//Eve: Stop time 1															@0000;2359;0000;2359;hhmm; ####
	CF9:INT;										//Holiday: Stop time 1														@0000;2359;0000;2359;hhmm; ####
	CF11:INT;									//Monday: Stop time 2														@0000;2359;0000;2359;hhmm; ####
	CF12:INT;									//Tuesday: Stop time 2													@0000;2359;0000;2359;hhmm; ####
	CF13:INT;									//Wednesday: Stop time 2												@0000;2359;0000;2359;hhmm; ####
	CF14:INT;									//Thursday: Stop time 2													@0000;2359;0000;2359;hhmm; ####
	CF15:INT;									//Friday: Stop time 2														@0000;2359;0000;2359;hhmm; ####
	CF16:INT;									//Saturday: Stop time 2													@0000;2359;0000;2359;hhmm; ####
	CF17:INT;									//Sunday: Stop time 2														@0000;2359;0000;2359;hhmm; ####
	CF18:INT;									//Eve: Stop time 2															@0000;2359;0000;2359;hhmm; ####
	CF19:INT;									//Holiday: Stop time 2														@0000;2359;0000;2359;hhmm; ####
	V:BOOL;										//Time channel is active
END_STRUCT
END_TYPE

// Device/AREA1/Struct/System/strManMode
TYPE strManMode :
STRUCT
	SP: DINT;									//Too long time in manual mode										@0;9999;0;9999;min; #### EU
	V: BOOL;									//Atleast one object in manual mode
	AL: BOOL;									//Long time in manual mode											@AL02
	ACK:BOOL;									//Acknowledge alarm
END_STRUCT
END_TYPE

// Device/AREA1/Struct/Sensors/strSensor7_Humidity
TYPE strSensor7_Humidity:
STRUCT
	PV:REAL;									//Process value																@-99;100;-99;100;°C; ###.# EU;T
	AD:DINT;									//Alarm Delay																@0;999;0;999;min; ### EU
	AL:BOOL;									//General alarm	
	FAULT:BOOL;								//Sensor error																	@AL02
	LAL:BOOL;									//Low alarm																	@AL02
	HAL:BOOL;									//High alarm																	@AL02
	ALL:REAL;									//Low alarm level															@-99;100;-99;100;°C; ###.# EU
	AHL:REAL;									//High alarm level															@-99;100;-99;100;°C; ###.# EU
	SP1:REAL;									//Minimum input value (scaling)										@0;100;0;100;%; ###.# EU
	SP2:REAL;									//Maximum input value (scaling)										@0;100;0;100;%; ###.# EU
	ACK:BOOL;									//Acknowledge alarm
	
	//Dewpoint
	CSP:REAL;									//Calculated setpoint for dewpoint									@-99;100;-99;100;°C; ###.# EU;T
	SP:REAL;									//Dewpoint offset															@-99;100;-99;100;°C; ###.# EU
	
	//Not used in Scada
	Symbol:INT;								//Symbol Value (0-3)
	Dew_En:BOOL;							//Enable function
END_STRUCT
END_TYPE

// Device/AREA1/Struct/Sensors/strSensor8_DefrostProtection
TYPE strSensor8_DefrostProtection :
STRUCT
	PV:REAL;									//Process value																@-99;100;-99;100;°C; ###.# EU;T
	AD:DINT;									//Alarm Delay																@0;999;0;999;min; ### EU
	AD1:DINT;									//Alarm Delay defrost														@0;9999;0;9999;min; #### EU
	AL:BOOL;									//General alarm	
	AL01:BOOL;									//Freeze protection activated											@AL02
	FAULT:BOOL;								//Sensor error																	@AL02
	LAL:BOOL;									//Low alarm																	@AL02
	HAL:BOOL;									//High alarm																	@AL02
	ALL:REAL;									//Low alarm level															@-99;100;-99;100;°C; ###.# EU
	AHL:REAL;									//High alarm level															@-99;100;-99;100;°C; ###.# EU
	SP1:REAL;									//Start temperature freeze protection								@-99;100;-99;100;°C; ###.# EU
	SP2:REAL;									//Stop temperature freeze protection								@-99;100;-99;100;°C; ###.# EU
	ACK:BOOL;									//Acknowledge alarm

	//Not used in Scada
	Symbol:INT;								//Symbol Value (0-3)
END_STRUCT
END_TYPE

// Device/AREA1/Struct/Sensors/strSensor9_CO2
TYPE strSensor9_CO2 :
STRUCT
	PV:REAL;									//Process value																@-99;100;-99;100;°C; ###.# EU;T
	AD:DINT;									//Alarm Delay																@0;999;0;999;min; ### EU
	AL:BOOL;									//General alarm	
	FAULT:BOOL;								//Sensor error																	@AL02
	LAL:BOOL;									//Low alarm																	@AL02
	HAL:BOOL;									//High alarm																	@AL02
	C02_HAL:BOOL;							//High carbon dioxide (CO2) content									@AL02
	HighAlarm:BOOL;							//CO2 Larmsignal															@AL02
	HL:REAL;									//High levels of air quality 												@0;9999;0;9999;ppm; #### EU
	LL:REAL;									//Low levels of air quality												@0;9999;0;9999;ppm; #### EU
	MAX1:REAL;								//Maximum degree of opening of the air damper					@0;100;0;100;%; ### EU
	MIN1:REAL;								//Minimum degree of opening of the air damper					@0;100;0;100;%; ### EU
	SP1:REAL;									//Minimum input value (scaling)										@0;9999;0;9999;ppm; #### EU
	SP2:REAL;									//Maximum input value (scaling)										@0;9999;0;9999;ppm; #### EU
	ACK:BOOL;									//Acknowledge alarm

	//Not used in Scada
	Symbol:INT;								//Symbol Value (0-3)
END_STRUCT
END_TYPE

// Device/AREA1/Struct/Functions/strFunction_Overtime
TYPE strFunction_Overtime :
STRUCT
	PV:INT;										//Time left																	@0;9999;0;9999;min; #### EU
	SP:INT;										//Set overtime																@0;9999;0;9999;min; #### EU
	V:BOOL;										//Overtime activated														@
	CMD:BOOL;									//Overtime

	//Not used in Scada
	En:BOOL;									//Enable function
END_STRUCT
END_TYPE

// Device/AREA1/Struct/Sensors/strSensor10_HeatExchanger_Pressure
TYPE strSensor10_HeatExchanger_Pressure :
STRUCT
	AL:BOOL;									//General alarm	
	InputAlarm:BOOL;						//Alarm signal
	HAL:BOOL;									//High differential pressure												@AL02
	ACK:BOOL;									//Acknowledge alarm

	//Not used in Scada
	Symbol:INT;								//Symbol Value (0-3)
END_STRUCT
END_TYPE

// Device/AREA1/Struct/Functions/strFunction_NightCooling
TYPE strFunction_NightCooling :
STRUCT
	SP1:REAL;									//Start value room temperature										@-99;100;-99;100;°C; ###.# EU
	SP2:REAL;									//Start value outdoor temperature										@-99;100;-99;100;°C; ###.# EU
	SP3:REAL;									//Stop value room temperature											@-99;100;-99;100;°C; ###.# EU
	SP4:REAL;									//Stop value outdoor temperature										@-99;100;-99;100;°C; ###.# EU
	SP5:REAL;									//Start value differential room-outdoor								@0;100;0;100;°C; ###.# EU
	SP6:REAL;									//Delayed night cooling 													@0;9999;0;9999;min; #### EU
	V:BOOL;										//Night cooling is activated												@
	V1:BOOL;									//Night cooling is blocked												@
	
	//Time Channel
	Arr:ARRAY [0..17] OF INT;
	CT1:INT;										//Monday: Start time 1													@0000;2359;0000;2359;hhmm; ####
	CT2:INT;										//Tuesday: Start time 1													@0000;2359;0000;2359;hhmm; ####
	CT3:INT;										//Wednesday: Start time 1												@0000;2359;0000;2359;hhmm; ####
	CT4:INT;										//Thursday: Start time 1													@0000;2359;0000;2359;hhmm; ####
	CT5:INT;										//Friday: Start time 1														@0000;2359;0000;2359;hhmm; ####
	CT6:INT;										//Saturday: Start time 1													@0000;2359;0000;2359;hhmm; ####
	CT7:INT;										//Sunday: Start time 1														@0000;2359;0000;2359;hhmm; ####
	CT8:INT;										//Eve: Start time 1															@0000;2359;0000;2359;hhmm; ####
	CT9:INT;										//Holiday: Start time 1													@0000;2359;0000;2359;hhmm; ####
	CF1:INT;										//Monday: Stop time 1														@0000;2359;0000;2359;hhmm; ####
	CF2:INT;										//Tuesday: Stop time 1													@0000;2359;0000;2359;hhmm; ####
	CF3:INT;										//Wednesday: Stop time 1												@0000;2359;0000;2359;hhmm; ####
	CF4:INT;										//Thursday: Stop time 1													@0000;2359;0000;2359;hhmm; ####
	CF5:INT;										//Friday: Stop time 1														@0000;2359;0000;2359;hhmm; ####
	CF6:INT;										//Saturday: Stop time 1													@0000;2359;0000;2359;hhmm; ####
	CF7:INT;										//Sunday: Stop time 1														@0000;2359;0000;2359;hhmm; ####
	CF8:INT;										//Eve: Stop time 1															@0000;2359;0000;2359;hhmm; ####
	CF9:INT;										//Holiday: Stop time 1														@0000;2359;0000;2359;hhmm; ####
	V2:BOOL;									//Time channel is active

	//Not used in Scada
	En:BOOL;									//Enable function
END_STRUCT
END_TYPE

// Device/AREA1/Struct/Functions/strFunction_NightHeating
TYPE strFunction_NightHeating :
STRUCT
	SP1:REAL;									//Start value room temperature										@-99;100;-99;100;°C; ###.# EU
	SP2:REAL;									//Start value outdoor temperature										@-99;100;-99;100;°C; ###.# EU
	SP3:REAL;									//Stop value room temperature											@-99;100;-99;100;°C; ###.# EU
	SP5:REAL;									//Delayed night heating 													@0;9999;0;9999;min; #### EU
	V:BOOL;										//Night heating is activated												@
	V1:BOOL;									//Night heating is blocked												@

	//Not used in Scada
	En:BOOL;									//Enable function
END_STRUCT
END_TYPE

// Device/AREA1/Struct/IO_Crevis/strST2792
TYPE strST2792 :
STRUCT
	ST2792_DO1:BOOL;						//Digital output 1
	ST2792_DO2:BOOL;						//Digital output 2
	ST2792_Switch1DI1:BOOL;				//Switch 1 Digital input 1
	ST2792_Switch1DI2:BOOL;				//Switch 1 Digital input 2
	ST2792_Switch2DI1:BOOL;				//Switch 2 Digital input 1
	ST2792_Switch2DI2:BOOL;				//Switch 2 Digital input 2
END_STRUCT
END_TYPE

// Device/AREA1/Struct/IO_Crevis/strST4491
TYPE strST4491 :
STRUCT
	ST4491_AO1:INT;							//Analog output 1
	ST4491_Switch1DI1:BOOL;				//Switch 1 Digital input 1
	ST4491_Switch2AI1:INT;				//Switch 2 Analog input 1
END_STRUCT
END_TYPE

// Device/AREA1/Struct/IO_Crevis/strST1218
TYPE strST1218 :
STRUCT
	ST1218_DI1:BOOL;						//Digital input 1
	ST1218_DI2:BOOL;						//Digital input 2
	ST1218_DI3:BOOL;						//Digital input 3
	ST1218_DI4:BOOL;						//Digital input 4
	ST1218_DI5:BOOL;						//Digital input 5
	ST1218_DI6:BOOL;						//Digital input 6
	ST1218_DI7:BOOL;						//Digital input 7
	ST1218_DI8:BOOL;						//Digital input 8
END_STRUCT
END_TYPE

// Device/AREA1/Struct/IO_Crevis/strST3708
TYPE strST3708 :
STRUCT
	ST3708_AI1:INT;							//RTD 1
	ST3708_AI2:INT;							//RTD 2
	ST3708_AI3:INT;							//RTD 3
	ST3708_AI4:INT;							//RTD 4
	ST3708_AI5:INT;							//RTD 5
	ST3708_AI6:INT;							//RTD 6
	ST3708_AI7:INT;							//RTD 7
	ST3708_AI8:INT;							//RTD 8
END_STRUCT
END_TYPE

// Device/AREA1/Struct/Units/strUC
TYPE strUC :
STRUCT
	//Sensors
	GT1:strSensor3_RegOutsideCompensation;				//Controlled temperature sensor with outsidecompenstation
	GT2:strSensor1;													//Measured sensor
	
	//Pumps
	P1:strPumpExercise;											//Heat pump
	
	//Valves
	SV1:strValveExercise;											//Heat valve
	
	//Misc signals
	GeneralStart:BOOL;												//UC started								@
	ManMode:strManMode;										//Alarm when one or more objects are in manual mode too long
	SWITCH:INT;														//Switch for the air unit		0=Off, 1=Manual, 2=Auto
END_STRUCT
END_TYPE

// Device/AREA1/Struct/HeatExchangers/strHeatExchanger_Cross
TYPE strHeatExchanger_Cross :
STRUCT
	AUT:INT;									//0=Auto, 1=Off, 2=On														@
	OP:REAL;									//Output value																@0;100;0;100;%; ### EU;T
	OPM:REAL;									//Manual output																@0;100;0;100;%; ###.# EU
	V:BOOL;										// On/Open																	@
	AL:BOOL;									//General alarm
	ACK:BOOL;									//Acknowledge alarm
	SP1:REAL;									//The opening degree when alarm										@0;100;0;100;%; ### EU
	SP2:DINT;									//Time open after alarm													@0;9999;0;9999;min; #### EU

	//Verkningsgradsberäkning
	PV1:REAL;									//Calculated efficiency													@0;100;0;100;%; ### EU;T
	AD:DINT;									//Efficiency, Alarm delay													@0;9999;0;9999;min; #### EU
	ALL:REAL;									//Efficiency, Alarm level 													@0;100;0;100;%; ###.# EU
	LAL:BOOL;									//Low efficiency																@AL02
	AL01:BOOL;									//Efficiency alarm
	
	//Kylåtervinning
	V01:BOOL;									//Cooling recovery activated												@
	SP3:REAL;									//Temperature difference for cooling recovery					@0;100;0;100;°C; ###.# EU
	
	//Preheating
	OP01:REAL;								//Calculated preheating value											@-99;100;-99;100;min; ###.# EU
	SP4:DINT;									//Preheating time															@0;9999;0;9999;min; #### EU
	SP5:REAL;									//The lowest outdoor temperature for preheating				@-99;100;-99;100;min; ###.# EU
	SP6:REAL;									//The highest outdoor temperature for preheating				@-99;100;-99;100;min; ###.# EU
	V02:BOOL;									//Preheating activated														@
	
	//Hardware switches
	ST2792_M:BOOL;							//Manual operating mode from hardware
	ST2792_MCMD:BOOL;					//Manual commanded starting from hardware
	ST4491_M:BOOL;							//Manual mode for analog value from hardware
	ST4491_OPM:REAL;						//Manual output value from hardware
	
	//Not used in Scada
	Symbol:INT;								//Symbol Value (0-3)
	Symbol_M:INT;							//Symbol in manual mode
	Seq_Heating:REAL;						//Control range of heat recovery
	Seq_Cooling:REAL;						//Control range for cooling recovery
	Eff_En:BOOL;								//Enable function
	CoolingRecycling_En:BOOL;			//Enable function
	Preheating_En:BOOL;					//Enable function
END_STRUCT
END_TYPE

// Device/AREA1/Struct/Dampers/strDamper_Analog
TYPE strDamper_Analog :
STRUCT
	CMD:BOOL;									//Command open															@
	OP:REAL;									//Process value																@0;100;0;100;%; ### EU;T
	AUT:INT;									//0=Auto, 1=Off, 2=On														@
	OPM:REAL;									//Manual output																@0;100;0;100;%; ###.# EU
	V:BOOL;										// On/Open																	@
	
	//Hardware switches
	ST2792_M:BOOL;							//Manual operating mode from hardware
	ST2792_MCMD:BOOL;					//Manual commanded starting from hardware
	ST4491_M:BOOL;							//Manual mode for analog value from hardware
	ST4491_OPM:REAL;						//Manual output value from hardware
	
	//Not used in Scada
	Symbol_M:INT;							//Symbol in manual mode
	StatusOff:BOOL;							//Stopped in manual mode
	StatusOn:BOOL;							//Started in manual mode
END_STRUCT
END_TYPE

// Device/AREA1/Struct/Pumps/strPumpExercise
TYPE strPumpExercise :
STRUCT
	AL:BOOL;									//General alarm																@
	AL01:BOOL;									//Feedback error																@AL01
	AL02:BOOL;									//Thermal relay triggered													@AL01
	CMD:BOOL;									//Commanded start															@;T
	AUT:INT;									//0=Auto, 1=Off, 2=On														@
	SP1:REAL;									//Start value SV																@0;100;0;100;%; ###.# EU
	SP2:REAL;									//Stop value SV																@0;100;0;100;%; ###.# EU
	SP3:DINT;									//Up time 																		@0;9999;0;9999;min; #### EU
	SP4:INT;										//Number of days before exercise										@0;999;0;999;dag; ### EU
	SP5:INT;										//Number of hours before exercise									@0;23;0;23;tim; ## EU
	ACK:BOOL;									//Acknowledge alarm

	//Misc parameters
	SP6:DINT;									//Feedback alarm delay													@0;3200;0;3200;s; #### EU
	SP7:REAL;									//Start value outdoor temperature										@-99;100;-99;100;°C; ###.# EU
	SP8:DINT;									//Thermal Relay alarm delay											@0;3200;0;3200;s; #### EU
	V:BOOL;										//On/Open																		@
	
	//Operating Time
	PV1:DINT;									//Total operating hours													@0;9999999;0;9999999;tim; ####### EU
	PV2:INT;										//Total operating minutes 												@0;59;0;59;min; ## EU	
	PV3:DINT;									//Total number of starts since reset									@0;9999999;0;9999999;st; ####### EU
	RST:BOOL;									//Resetting the operation time and number of starts			@
	
	//Excercise
	PV4:INT;										//Days before exercise														@0;999;0;999;dag; ### EU
	PV5:INT;										//Hours before exercise													@0;23;0;23;tim; ## EU
	PV6:INT;										//Minutes before exercise 												@0;59;0;59;min; ## EU	
	SP9:INT;										//Starting day exercise														@0;6;0;6;dag; # EU
	SP10:INT;									//Starting time exercise													@0;23;0;23;tim; ## EU
	SP11:INT;									//Starting time exercise 													@0;59;0;59;min; ## EU
	SP12:INT;									//Exercise time 																@0;999;0;999;min; ### EU
	V01:BOOL;									//Status exercise																@
		
	//Hardware switches
	ST2792_M:BOOL;							//Manual operating mode from hardware
	ST2792_MCMD:BOOL;					//Manual commanded starting from hardware
	ST4491_M:BOOL;							//Manual mode for analog value from hardware
	ST4491_OPM:REAL;						//Manual output value from hardware
		
	//Not used in Scada
	Symbol:INT;								//Symbol Value (0-3)
	Symbol_M:INT;							//Symbol in manual mode
	ManualStatusOff:BOOL;				//Stopped in manual mode
	ManualStatusOn:BOOL;					//Started in manual mode
	EnFeedbackError:BOOL;				//Activate feedback alarm
	FeedbackError:BOOL;					//Feedback error
	EnTempControl:BOOL;					//Activate temperature control	
	EnThermalError:BOOL;					//Activate Thermal Relay alarm
	ThermalError:BOOL;						//Thermal relay triggered
	ThermicRelay:BOOL;					//Feedback thermo relay	
	Ex_En:BOOL;								//Enable exercise
	Ex_En_Day:BOOL;							//Enable specific day
	Ex_En_Time:BOOL;						//Enable specific time	
	Ex_SecOff:DINT;							//Enumeration of seconds when the object is not in operation
	Ex_SavedData:ARRAY [0..3] OF INT;//Saved data for the object			
END_STRUCT
END_TYPE

// Device/AREA1/Struct/Valves/strValve
TYPE strValve :
STRUCT
	AUT:INT;									//0=Auto, 1=Off, 2=On														@
	OP:REAL;									//Output value																@0;100;0;100;%; ### EU;T
	OPM:REAL;									//Manual output																@0;100;0;100;%; ###.# EU
	V:BOOL;										// On/Open																	@
	
	//Hardware switches
	ST2792_M:BOOL;							//Manual operating mode from hardware
	ST2792_MCMD:BOOL;					//Manual commanded starting from hardware
	ST4491_M:BOOL;							//Manual mode for analog value from hardware
	ST4491_OPM:REAL;						//Manual output value from hardware

	//Not used in Scada
	Frost_V:BOOL;								//Antifreeze activated
	Frost_En:BOOL;							//Enable antifreeze
	Symbol_M:INT;							//Symbol in manual mode
	Seq_Output:REAL;						//Control range of valve
END_STRUCT
END_TYPE

// Device/AREA1/Struct/Pumps/strPump
TYPE strPump :
STRUCT
	AL:BOOL;									//General alarm																@
	AL01:BOOL;									//Feedback error																@AL01
	AL02:BOOL;									//Thermal relay triggered													@AL01
	CMD:BOOL;									//Commanded start															@;T
	AUT:INT;									//0=Auto, 1=Off, 2=On														@
	SP1:REAL;									//Start value SV																@0;100;0;100;%; ###.# EU
	SP2:REAL;									//Stop value SV																@0;100;0;100;%; ###.# EU
	SP3:DINT;									//Up time 																		@0;9999;0;9999;min; #### EU
	ACK:BOOL;									//Acknowledge alarm

	//Misc parameters
	SP6:DINT;									//Feedback alarm delay													@0;3200;0;3200;s; #### EU
	SP7:REAL;									//Start value outdoor temperature										@-99;100;-99;100;°C; ###.# EU
	SP8:DINT;									//Thermal Relay alarm delay											@0;3200;0;3200;s; #### EU
	V:BOOL;										//On/Open																		@
	
	//Operating Time
	PV1:DINT;									//Total operating hours													@0;9999999;0;9999999;tim; ####### EU
	PV2:INT;										//Total operating minutes 												@0;59;0;59;min; ## EU	
	PV3:DINT;									//Total number of starts since reset    								@0;9999999;0;9999999;st; ####### EU
	RST:BOOL;									//Resetting the operation time and number of starts			@
	
	//Hardware switches
	ST2792_M:BOOL;							//Manual operating mode from hardware
	ST2792_MCMD:BOOL;					//Manual commanded starting from hardware
	ST4491_M:BOOL;							//Manual mode for analog value from hardware
	ST4491_OPM:REAL;						//Manual output value from hardware
		
	//Not used in Scada
	Symbol:INT;								//Symbol Value (0-3)
	Symbol_M:INT;							//Symbol in manual mode
	ManualStatusOff:BOOL;				//Stopped in manual mode
	ManualStatusOn:BOOL;					//Started in manual mode
	EnFeedbackError:BOOL;				//Activate feedback alarm
	FeedbackError:BOOL;					//Feedback error
	EnTempControl:BOOL;					//Activate temperature control	
	EnThermalError:BOOL;					//Activate Thermal Relay alarm
	ThermalError:BOOL;						//Thermal relay triggered
	ThermicRelay:BOOL;					//Feedback thermo relay	
END_STRUCT
END_TYPE

// Device/AREA1/Struct/System/strSummerTime
TYPE strSummerTime :
STRUCT
	AverageTempCheck_En: BOOL;						//Temperature control enable
	AverageTempSummer: REAL;							//Average temperaute value for the summer period
	AverageTempWinter: REAL;							//Average temperaute value for the winter period
	LowOutsideTemp: REAL;								//Lower temperature limit for the winter period
	NumberOfSummerDays: INT;							//Number of days before transition to summer period
	NumberOfWinterDays: INT;							//Number of days before transition TO winter period
	SummerMode_V: BOOL;								//Summer period is active
	SummerMonthCheck_En: BOOL;						//Month control is enable
	SummerMonthEnd: INT;								//Month when summer period is ending
	SummerMonthStart: INT;								//Month when summer period is starting
	TemperatureAverage: REAL;							//Actual average value for the outdoor temperature


	//Not used in Scada
	CounterSummerDays: INT;								//Internal counter
	CounterWinterDays: INT;								//Internal counter
	WorkingData: REAL;										//Saved working data
END_STRUCT
END_TYPE

// Device/AREA1/Struct/Fans/strFan_Onespeed
TYPE strFan_Onespeed :
STRUCT
	AUT:INT;									//0=Auto, 1=Off, 2=On														@
	AL:BOOL;									//General alarm
	AL01:BOOL;									//Feedback error																@AL01
	AL02:BOOL;									//Thermal relay triggered													@AL01
	V:BOOL;										// On/Open																	@
	CMD:BOOL;									//Commanded start															@
	SP1:DINT;									//Start delay																	@0;3200;0;3200;s; #### EU
	SP2:DINT;									//Thermal Relay alarm delay											@0;3200;0;3200;s; #### EU
	SP3:DINT;									//Fan guard alarm delay													@0;3200;0;3200;s; #### EU
	SP4:DINT;									//Feedback alarm delay													@0;3200;0;3200;s; #### EU
	ACK:BOOL;									//Acknowledge alarm

	//Operating Time
	PV1:DINT;									//Total operating hours													@0;9999999;0;9999999;tim; ####### EU
	PV2:INT;										//Total operating minutes 												@0;59;0;59;min; ## EU	
	PV3:DINT;									//Total number of starts since reset									@0;9999999;0;9999999;st; ####### EU
	RST:BOOL;									//Resetting the operation time and number of starts			@	
	
	//Hardware switches
	ST2792_M:BOOL;							//Manual operating mode from hardware
	ST2792_MCMD:BOOL;					//Manual commanded starting from hardware
	ST4491_M:BOOL;							//Manual mode for analog value from hardware
	ST4491_OPM:REAL;						//Manual output value from hardware
	
	//Not used in Scada
	Symbol:INT;								//Symbol Value (0-3)
	Symbol_M:INT;							//Symbol in manual mode
	Operating:BOOL;							//Objects in operation
	StatusOff:BOOL;							//Stopped in manual mode
	StatusOn:BOOL;							//Started in manual mode
	SumAlarm:BOOL;							//General alarm
	RunIndication:BOOL;					//Operating indicator
	ManualStart:BOOL;						//Manual start command
	EnFeedbackError:BOOL;				//Activate feedback alarm
	FeedbackError:BOOL;					//Feedback error
	EnThermalError:BOOL;					//Activate Thermal Relay alarm
	ThermalError:BOOL;						//Thermal relay fault
	EnFanGuardError:BOOL;				//Activate Fan Guard error
	FanGuardError:BOOL;					//Fan Guard error
	ThermoRelay1:BOOL;					//Thermal Relay ok, halfspeed
END_STRUCT
END_TYPE

// Device/AREA1/Struct/Sensors/strSensor11_DifferentialPressure
TYPE strSensor11_DifferentialPressure :
STRUCT
	V:BOOL;										//Status
	AD:DINT;									//Alarm Delay																@0;999;0;999;min; ### EU
	AL:BOOL;									//General alarm	
	HAL:BOOL;									//Filter guard alarm														@AL02
	ACK:BOOL;									//Acknowledge alarm

	//Not used in Scada
	Symbol:INT;								//Symbol Value (0-3)
END_STRUCT
END_TYPE

// Device/AREA1/B001/GVL_B001
VAR_GLOBAL
	SystemTags: strSystemTags;									//Systemtags
	SYS_StartupDelayComm:BOOL;								//Startup time for communication
	SYS_InitPulse:BOOL;												//Init pulse
	SYS_Pulse100ms:BOOL;											//100 ms pulse
	SYS_SecondPulse:BOOL;										//Second pulse
	SYS_MinutePulse:BOOL;										//Minute pulse
	SYS_ArrayPlcTime:ARRAY [0..6] OF INT;					//Date and Time

	AS_SWITCH_MAN21:BOOL;										//Switch in maual mode
	AS_SWITCH_AUT11:BOOL;										//Switch in auto mode

	ActivateModbus:BOOL; 										 //BARA FÖR TEST
		
	//IO
	InputArea:ARRAY [0..11] OF WORD;						//Input register
	OutputArea:ARRAY [0..1] OF WORD;						//Output register
	Nod1_Slot1:strST3708;											//Nod1 Slot1
	Nod1_Slot2:strST4491;											//Nod1 Slot2
	Nod1_Slot3:strST1218;											//Nod1 Slot3
	Nod1_Slot4:strST2792;											//Nod1 Slot4
END_VAR

// Device/AREA1/B001/B001
VAR_GLOBAL PERSISTENT RETAIN
	LB01:strLB;													//Tags associated with LB01
	UCSh1:strUC;												//Tags associated with UC Sh1
	AS_SWITCH:INT;											//Service switch on cabinet 0=Off, 1=Hand, 2=Auto
	SYS_E_AckAlarm:BOOL;									//Acknowledge all alarms
	SYS_Fire_AL:BOOL;										//Firealarm
	SYS_Fire_AlAck_AL:BOOL;								//Acknowledge alarm
	SYS_SWT:strSummerTime;								//Summer period
	SYS_Evening:BOOL;										//Evening flag
	SYS_Holiday:BOOL;										//Holiday flag
	SYS_HolidayDates:ARRAY [0..19] OF INT;	
	SYS_PLC_VersionNr: STRING(4);						//Version number on the application
	SYS_PLC_VersionDate: STRING(10);					//Date on the application
END_VAR

// Device/AREA1/System/Functions/Sys_SummerPeriod
PROGRAM Sys_SummerPeriod
VAR
	Control_SweHoliday: _BE_Holiday_Swe;
	Control_Holiday: _BE_Holiday;
	fb_SummerWinter: _BE_SummerWinterAverage;
END_VAR

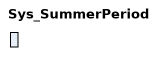
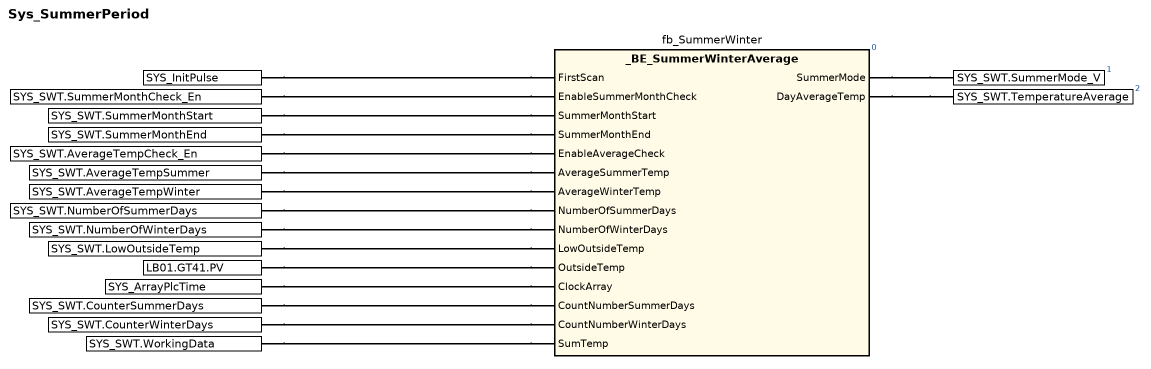
fb_SummerWinter(
    FirstScan := SYS_InitPulse,
    EnableSummerMonthCheck := SYS_SWT.SummerMonthCheck_En,
    SummerMonthStart := SYS_SWT.SummerMonthStart,
    SummerMonthEnd := SYS_SWT.SummerMonthEnd,
    EnableAverageCheck := SYS_SWT.AverageTempCheck_En,
    AverageSummerTemp := SYS_SWT.AverageTempSummer,
    AverageWinterTemp := SYS_SWT.AverageTempWinter,
    NumberOfSummerDays := SYS_SWT.NumberOfSummerDays,
    NumberOfWinterDays := SYS_SWT.NumberOfWinterDays,
    LowOutsideTemp := SYS_SWT.LowOutsideTemp,
    OutsideTemp := LB01.GT41.PV,
    ClockArray := SYS_ArrayPlcTime,
    CountNumberSummerDays := SYS_SWT.CounterSummerDays,
    CountNumberWinterDays := SYS_SWT.CounterWinterDays,
    SumTemp := SYS_SWT.WorkingData); // _BE_SummerWinterAverage
SYS_SWT.SummerMode_V := fb_SummerWinter.SummerMode;
SYS_SWT.TemperatureAverage := fb_SummerWinter.DayAverageTemp;

END_PROGRAM

// Device/AREA1/System/Functions/Sys_CalculateHoliday
PROGRAM Sys_CalculateHoliday
VAR
	Control_SweHoliday: _BE_Holiday_Swe;
	Control_Holiday: _BE_Holiday;
	fb_SummerWinter: _BE_SummerWinterAverage;
END_VAR

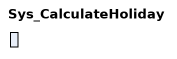
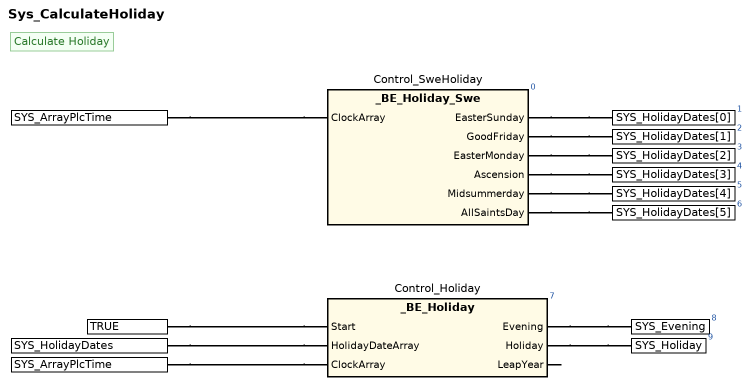
// Calculate Holiday
Control_SweHoliday(ClockArray := SYS_ArrayPlcTime); // _BE_Holiday_Swe
SYS_HolidayDates[0] := Control_SweHoliday.EasterSunday;
SYS_HolidayDates[1] := Control_SweHoliday.GoodFriday;
SYS_HolidayDates[2] := Control_SweHoliday.EasterMonday;
SYS_HolidayDates[3] := Control_SweHoliday.Ascension;
SYS_HolidayDates[4] := Control_SweHoliday.Midsummerday;
SYS_HolidayDates[5] := Control_SweHoliday.AllSaintsDay;
Control_Holiday(Start := TRUE, HolidayDateArray := SYS_HolidayDates, ClockArray := SYS_ArrayPlcTime); // _BE_Holiday
SYS_Evening := Control_Holiday.Evening;
SYS_Holiday := Control_Holiday.Holiday;

END_PROGRAM

// Device/AREA1/System/SystemSignals/Sys_SystemTags
PROGRAM Sys_SystemTags
VAR
	SystemSignals_FB: FB_SystemSignals;
	FbInitPulse: R_TRIG;
	Fb100msPulse: R_TRIG;
	Fb1sPulse: R_TRIG;
	Fb1mPulse: R_TRIG;
END_VAR
VAR // added by the converter: edge detectors and wires of the graphical bodies
    _w1 : BOOL;
    _w2 : ANY;
    _w3 : INT;
END_VAR

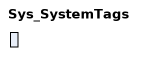
SystemSignals_FB(); // FB_SystemSignals
SystemTags.xAlwaysFalse := SystemSignals_FB.SysSignals.strSystemTags;
SystemTags.xAlwaysTrue := SystemSignals_FB.SysSignals.xAlwaysFalse;
SystemTags.xOnFirstScan := SystemSignals_FB.SysSignals.xAlwaysTrue;
SystemTags.xPulseMinute := SystemSignals_FB.SysSignals.xFlash100ms;
SystemTags.xPulse1s := SystemSignals_FB.SysSignals.xPulseMinute;
SystemTags.xPulse100ms := SystemSignals_FB.SysSignals.xPulse1s;
SystemTags.xCurrentTimeAndDate := SystemSignals_FB.SysSignals.xPulse100ms;
SystemTags.xNewDayPulse := SystemSignals_FB.SysSignals.xCurrentTimeAndDate;
// Actual PLC Time
SYS_ArrayPlcTime[6] := UINT_TO_INT(SystemTags.xCurrentTimeAndDate.wDayOfWeek);
_w1 := SystemTags.xCurrentTimeAndDate.wDayOfWeek = 7;
IF _w1 THEN _w2 := 0; END_IF
IF _w1 THEN _w3 := UINT_TO_INT(_w2); END_IF
SYS_ArrayPlcTime[6] := _w3;
SYS_ArrayPlcTime[0] := UINT_TO_INT(SystemTags.xCurrentTimeAndDate.RTS_SYSTIMEDATE);
SYS_ArrayPlcTime[1] := UINT_TO_INT(SystemTags.xCurrentTimeAndDate.wYear);
SYS_ArrayPlcTime[2] := UINT_TO_INT(SystemTags.xCurrentTimeAndDate.wMonth);
SYS_ArrayPlcTime[3] := UINT_TO_INT(SystemTags.xCurrentTimeAndDate.wDay);
SYS_ArrayPlcTime[4] := UINT_TO_INT(SystemTags.xCurrentTimeAndDate.wHour);
SYS_ArrayPlcTime[5] := UINT_TO_INT(SystemTags.xCurrentTimeAndDate.wMinute);
// Init pulse
FbInitPulse(CLK := SystemTags.xOnFirstScan); // R_TRIG
SYS_InitPulse := FbInitPulse.Q;
// 100 ms pulse
Fb100msPulse(CLK := SystemTags.xPulse100ms); // R_TRIG
SYS_Pulse100ms := Fb100msPulse.Q;
// Second pulse
Fb1sPulse(CLK := SystemTags.xPulse1s); // R_TRIG
SYS_SecondPulse := Fb1sPulse.Q;
// Minute pulse
Fb1mPulse(CLK := SystemTags.xPulseMinute); // R_TRIG
SYS_MinutePulse := Fb1mPulse.Q;

END_PROGRAM

// Device/AREA1/FB/FB_SystemSignals
FUNCTION_BLOCK FB_SystemSignals

VAR_OUTPUT
	SysSignals: strSystemTags;
END_VAR
VAR
	// RTC DateTime in Secounds
	dwActualTime: DWORD;
	// Daylight Compencated DateTime in secounds
	dwLocalTime: DWORD;
	SysTimeRTCGet_pResult: UDINT;
	latesthour: UINT;
	latestSecond: UINT;
	latestMin: UINT;
	flag: BOOL;
	cyclicCounter: INT;
	//blink100ms:BLINK;
	pulse100ms: INT;
END_VAR

//Always False Signal
SysSignals.xAlwaysFalse := FALSE;

//Always True
SysSignals.xAlwaysTrue := TRUE;

//On first scan
IF NOT flag THEN
	SysSignals.xOnFirstScan := TRUE;
ELSE
	SysSignals.xOnFirstScan := FALSE;
END_IF
flag := TRUE;

//Read Time from 1970 in seconds
dwActualTime := SysTimeRtcGet(pResult:=SysTimeRTCGet_pResult);
//Convert this second from UTC to Date and time compensated
SysTimeRtcConvertUtcToLocal(dwTimestampUtc:=dwActualTime, pdwTimestampLocal:=dwLocalTime);
//Convert to date time format
SysTimeRtcConvertUtcToDate(dwTimestampUtc:=dwLocalTime, pDate:=SysSignals.xCurrentTimeAndDate);

//New Day pulse
IF latesthour = 23 AND SysSignals.xCurrentTimeAndDate.wHour = 0 THEN
	SysSignals.xNewDayPulse := TRUE;
ELSE
	SysSignals.xNewDayPulse := FALSE;
END_IF
latesthour := SysSignals.xCurrentTimeAndDate.wHour;

//Second pulse
IF latestSecond <> SysSignals.xCurrentTimeAndDate.wSecond THEN
	SysSignals.xPulse1s := TRUE;
ELSE
	SysSignals.xPulse1s := FALSE;	
END_IF
latestSecond := SysSignals.xCurrentTimeAndDate.wSecond;

//Minute pulse
IF latestMin <> SysSignals.xCurrentTimeAndDate.wMinute THEN
	SysSignals.xPulseMinute:=TRUE;
ELSE
	SysSignals.xPulseMinute:=FALSE;
END_IF
latestMin := SysSignals.xCurrentTimeAndDate.wMinute;

//100ms pulse
//blink100ms(ENABLE:=TRUE, TIMELOW:=T#50MS, TIMEHIGH:=T#50MS);
//pulse100ms(CLK:=blink100ms.OUT, Q=>SysSignals.xPulse100ms);

//100 ms pulse if task is 20 ms
IF cyclicCounter>=5 THEN
	SysSignals.xPulse100ms:=TRUE;
	cyclicCounter:=1;
ELSE
	cyclicCounter:=cyclicCounter+1;
	SysSignals.xPulse100ms:=FALSE;	
END_IF

END_FUNCTION_BLOCK

// Device/AREA1/System/Communication/Sys_StartUp
PROGRAM Sys_StartUp
VAR
	delayStartUpTimer: TON;
END_VAR

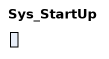
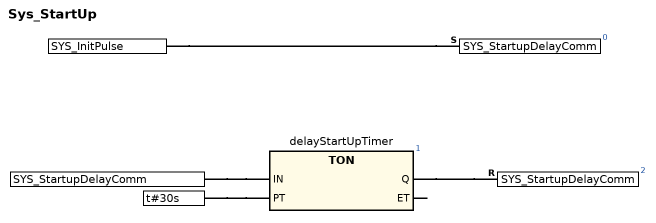
SYS_StartupDelayComm S= SYS_InitPulse;
delayStartUpTimer(IN := SYS_StartupDelayComm, PT := t#30s); // TON
SYS_StartupDelayComm R= delayStartUpTimer.Q;

END_PROGRAM

// Device/AREA1/System/Communication/Sys_CommunicationAlarm
PROGRAM Sys_CommunicationAlarm
VAR
	fb_nod1: R_TRIG;
	fb_nod2: R_TRIG;
	fb_nod3: R_TRIG;
	fb_TON_reset: TON;
END_VAR
VAR // added by the converter: edge detectors and wires of the graphical bodies
    _w1 : ANY;
END_VAR

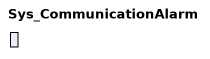
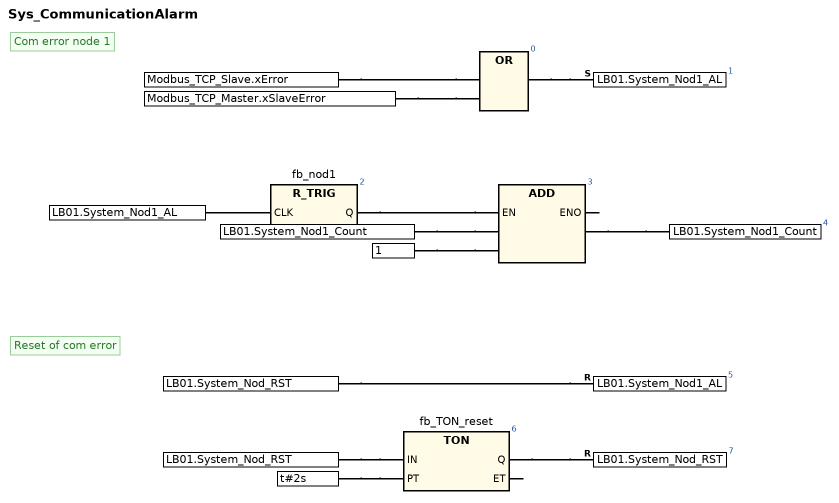
// Com error node 1
LB01.System_Nod1_AL S= Modbus_TCP_Slave.xError OR Modbus_TCP_Master.xSlaveError;
fb_nod1(CLK := LB01.System_Nod1_AL); // R_TRIG
IF fb_nod1.Q THEN _w1 := LB01.System_Nod1_Count + 1; END_IF
LB01.System_Nod1_Count := _w1;
LB01.System_Nod1_AL R= LB01.System_Nod_RST;
// Reset of com error
fb_TON_reset(IN := LB01.System_Nod_RST, PT := t#2s); // TON
LB01.System_Nod_RST R= fb_TON_reset.Q;

END_PROGRAM

// Device/AREA1/B001/LB01/AirHandlingUnit/LB01_Alarm
PROGRAM LB01_Alarm
VAR
	fb_nod1: R_TRIG;
	fb_TON_reset: TON;
	AlarmAcknowledge01: _BE_AlarmAckRemote;
	timerManMode: TON;
	_BE_AlarmAckRemote_0: _BE_AlarmAckRemote;
END_VAR
VAR // added by the converter: edge detectors and wires of the graphical bodies
    _w1 : TIME;
    _w2 : BOOL;
END_VAR

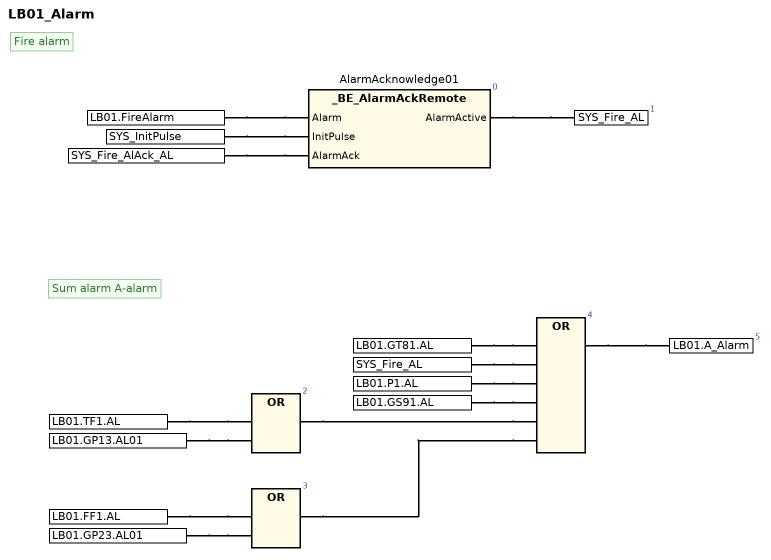
// Fire alarm
AlarmAcknowledge01(Alarm := LB01.FireAlarm, InitPulse := SYS_InitPulse, AlarmAck := SYS_Fire_AlAck_AL); // _BE_AlarmAckRemote
SYS_Fire_AL := AlarmAcknowledge01.AlarmActive;
// Sum alarm A-alarm
LB01.A_Alarm := LB01.GT81.AL OR SYS_Fire_AL OR LB01.P1.AL OR LB01.GS91.AL OR (LB01.TF1.AL OR LB01.GP13.AL01) OR (LB01.FF1.AL OR LB01.GP23.AL01);
_w1 := DINT_TO_TIME(LB01.ManMode.SP * 60000);
_w2 := LB01.P1.AUT > 0 OR LB01.P2.AUT > 0 OR LB01.ST11.AUT > 0 OR LB01.ST21.AUT > 0 OR LB01.TF1.AUT > 0 OR LB01.FF1.AUT > 0 OR LB01.SV61.AUT > 0 OR LB01.SV62.AUT > 0 OR LB01.GT11.M OR LB01.GT31.M OR LB01.GT11_Cool.M;
LB01.ManMode.V := _w2;
timerManMode(IN := _w2, PT := _w1); // TON
_BE_AlarmAckRemote_0(Alarm := timerManMode.Q, InitPulse := SYS_InitPulse, AlarmAck := LB01.ManMode.ACK); // _BE_AlarmAckRemote
LB01.ManMode.AL := _BE_AlarmAckRemote_0.AlarmActive;

END_PROGRAM

// Device/AREA1/B001/LB01/AirHandlingUnit/LB01_StartConditions
PROGRAM LB01_StartConditions
VAR

END_VAR
VAR // added by the converter: edge detectors and wires of the graphical bodies
    _w1, _w2, _w3 : ANY;
END_VAR

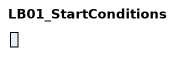
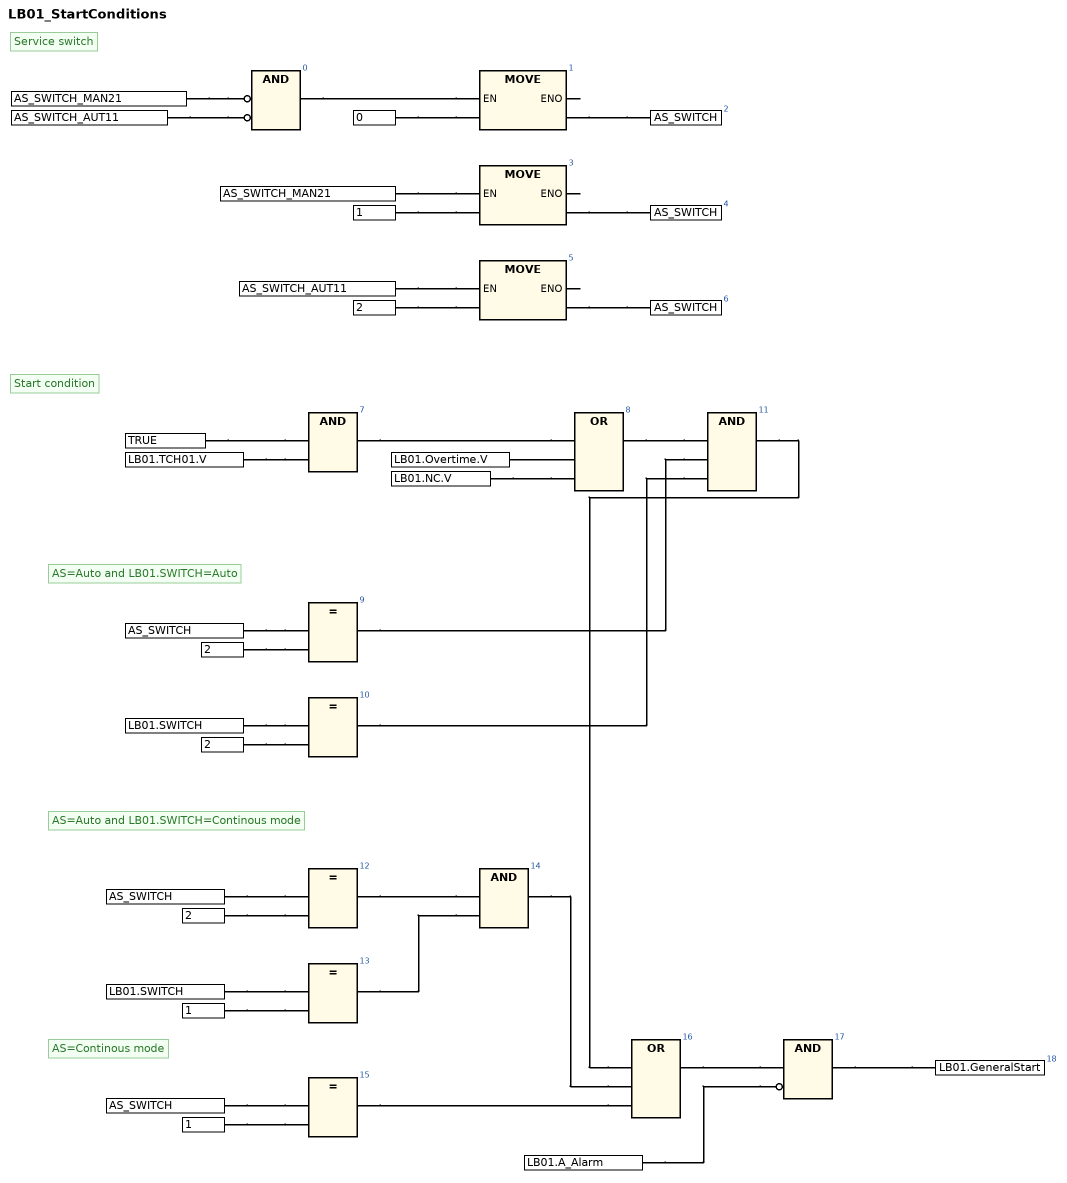
// Service switch
IF NOT AS_SWITCH_MAN21 AND NOT AS_SWITCH_AUT11 THEN _w1 := 0; END_IF
AS_SWITCH := _w1;
IF AS_SWITCH_MAN21 THEN _w2 := 1; END_IF
AS_SWITCH := _w2;
IF AS_SWITCH_AUT11 THEN _w3 := 2; END_IF
AS_SWITCH := _w3;
// Start condition
// AS=Auto and LB01.SWITCH=Auto
// AS=Auto and LB01.SWITCH=Continous mode
// AS=Continous mode
LB01.GeneralStart := ((TRUE AND LB01.TCH01.V OR LB01.Overtime.V OR LB01.NC.V) AND AS_SWITCH = 2 AND LB01.SWITCH = 2 OR AS_SWITCH = 2 AND LB01.SWITCH = 1 OR AS_SWITCH = 1) AND NOT LB01.A_Alarm;

END_PROGRAM

// Device/AREA1/B001/LB01/AirHandlingUnit/LB01_TimeChannel
PROGRAM LB01_TimeChannel
VAR
	Control_TimeChannel1: _BE_TimeChannel_CiFAS;
	Control_TimeChannel_NC: _BE_TimeChannel_CiFAS;
END_VAR

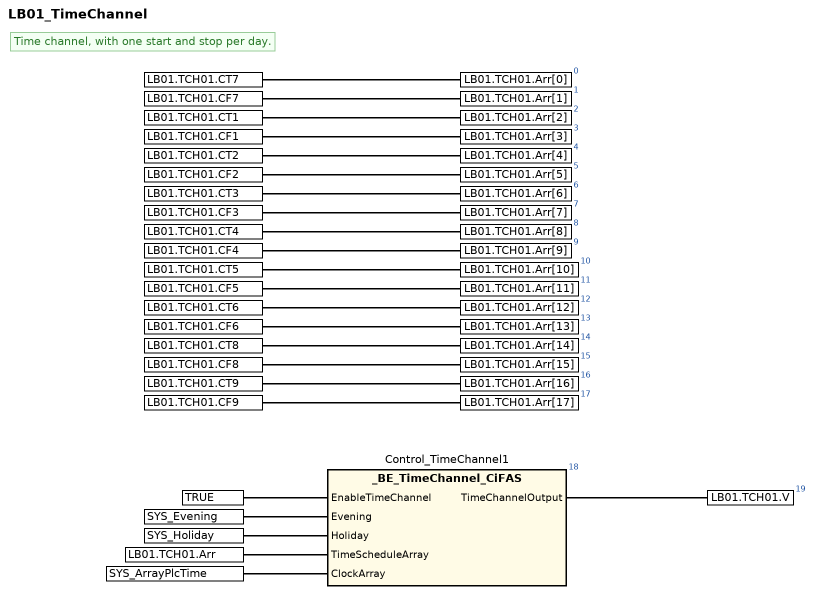
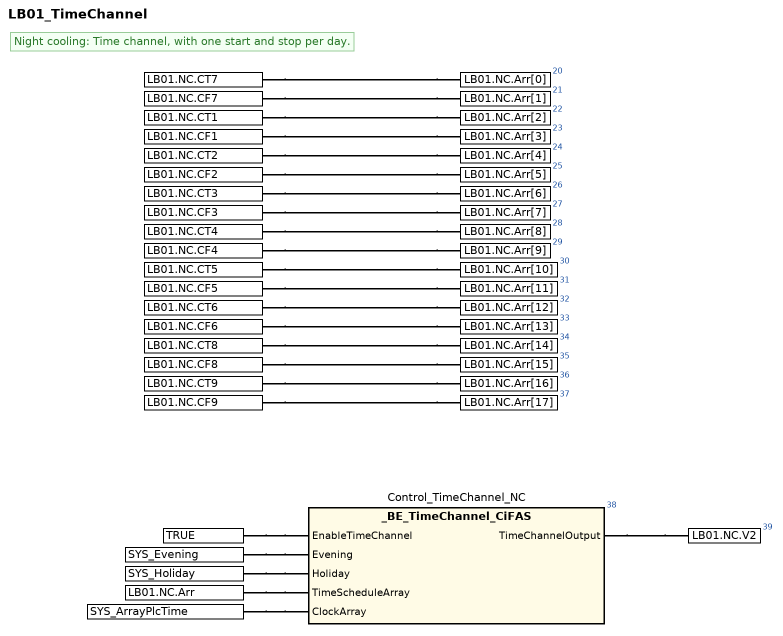
// Time channel, with one start and stop per day.
LB01.TCH01.Arr[0] := LB01.TCH01.CT7;
LB01.TCH01.Arr[1] := LB01.TCH01.CF7;
LB01.TCH01.Arr[2] := LB01.TCH01.CT1;
LB01.TCH01.Arr[3] := LB01.TCH01.CF1;
LB01.TCH01.Arr[4] := LB01.TCH01.CT2;
LB01.TCH01.Arr[5] := LB01.TCH01.CF2;
LB01.TCH01.Arr[6] := LB01.TCH01.CT3;
LB01.TCH01.Arr[7] := LB01.TCH01.CF3;
LB01.TCH01.Arr[8] := LB01.TCH01.CT4;
LB01.TCH01.Arr[9] := LB01.TCH01.CF4;
LB01.TCH01.Arr[10] := LB01.TCH01.CT5;
LB01.TCH01.Arr[11] := LB01.TCH01.CF5;
LB01.TCH01.Arr[12] := LB01.TCH01.CT6;
LB01.TCH01.Arr[13] := LB01.TCH01.CF6;
LB01.TCH01.Arr[14] := LB01.TCH01.CT8;
LB01.TCH01.Arr[15] := LB01.TCH01.CF8;
LB01.TCH01.Arr[16] := LB01.TCH01.CT9;
LB01.TCH01.Arr[17] := LB01.TCH01.CF9;
Control_TimeChannel1(
    EnableTimeChannel := TRUE,
    Evening := SYS_Evening,
    Holiday := SYS_Holiday,
    TimeScheduleArray := LB01.TCH01.Arr,
    ClockArray := SYS_ArrayPlcTime); // _BE_TimeChannel_CiFAS
LB01.TCH01.V := Control_TimeChannel1.TimeChannelOutput;
// Night cooling: Time channel, with one start and stop per day.
LB01.NC.Arr[0] := LB01.NC.CT7;
LB01.NC.Arr[1] := LB01.NC.CF7;
LB01.NC.Arr[2] := LB01.NC.CT1;
LB01.NC.Arr[3] := LB01.NC.CF1;
LB01.NC.Arr[4] := LB01.NC.CT2;
LB01.NC.Arr[5] := LB01.NC.CF2;
LB01.NC.Arr[6] := LB01.NC.CT3;
LB01.NC.Arr[7] := LB01.NC.CF3;
LB01.NC.Arr[8] := LB01.NC.CT4;
LB01.NC.Arr[9] := LB01.NC.CF4;
LB01.NC.Arr[10] := LB01.NC.CT5;
LB01.NC.Arr[11] := LB01.NC.CF5;
LB01.NC.Arr[12] := LB01.NC.CT6;
LB01.NC.Arr[13] := LB01.NC.CF6;
LB01.NC.Arr[14] := LB01.NC.CT8;
LB01.NC.Arr[15] := LB01.NC.CF8;
LB01.NC.Arr[16] := LB01.NC.CT9;
LB01.NC.Arr[17] := LB01.NC.CF9;
Control_TimeChannel_NC(
    EnableTimeChannel := TRUE,
    Evening := SYS_Evening,
    Holiday := SYS_Holiday,
    TimeScheduleArray := LB01.NC.Arr,
    ClockArray := SYS_ArrayPlcTime); // _BE_TimeChannel_CiFAS
LB01.NC.V2 := Control_TimeChannel_NC.TimeChannelOutput;

END_PROGRAM

// Device/AREA1/B001/LB01/Sensor/Temperature/GT81/LB01_GT81
PROGRAM LB01_GT81
VAR
	local:strSensor5_FreezeProtection;
	alack_al01: BOOL;
	FbFreezeProt: _BE_ReturnWaterControl;
	gt_Min: TON;
	gt_Max: TON;
	ackFault: BOOL;
	ackLal: BOOL;
	ackHal: BOOL;
	ackAl01: BOOL;
	AlarmAcknowledge01: _BE_AlarmAckRemote;
	AlarmAcknowledge02: _BE_AlarmAckRemote;
	AlarmAcknowledge03: _BE_AlarmAckRemote;
	AlarmFb01: _BE_AlarmAckRequired;
END_VAR
VAR // added by the converter: edge detectors and wires of the graphical bodies
    _w1, _w2, _w3 : ANY;
END_VAR

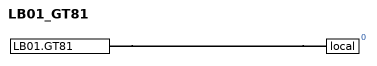
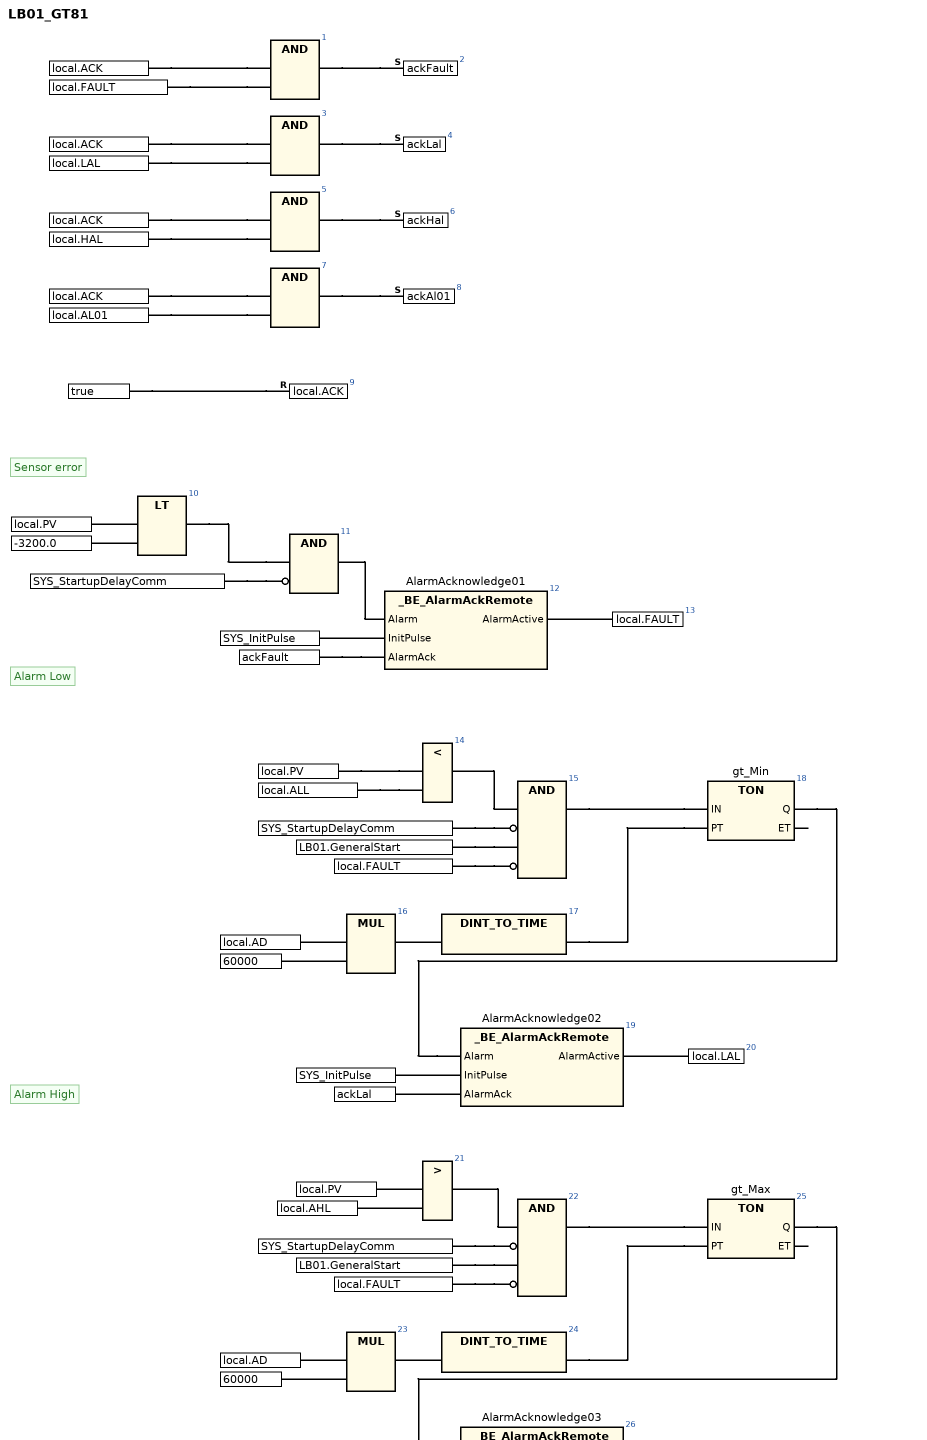
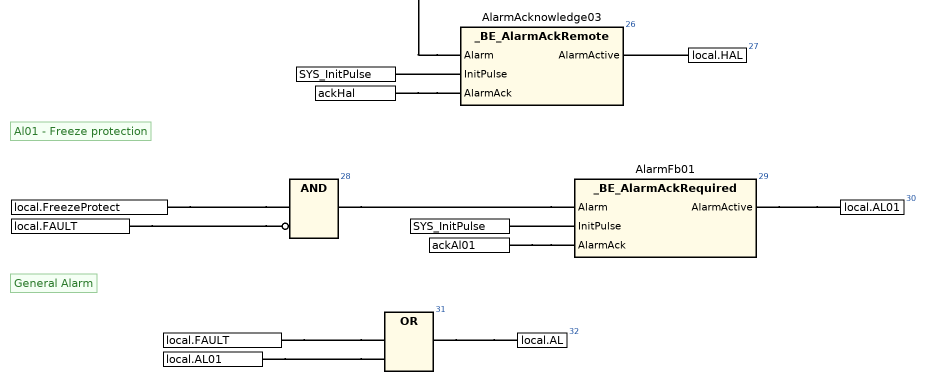
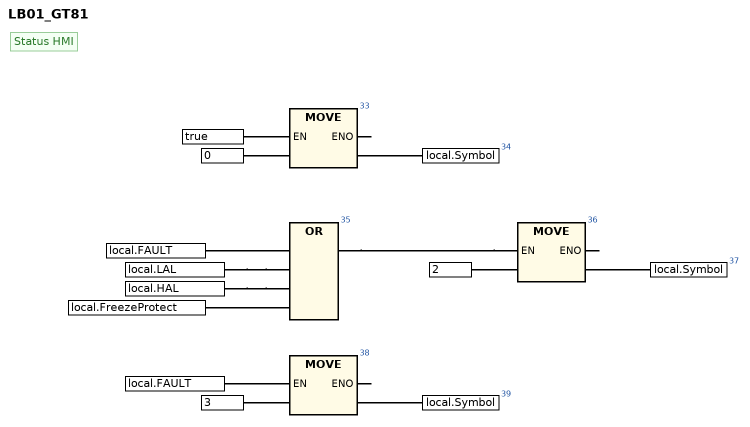
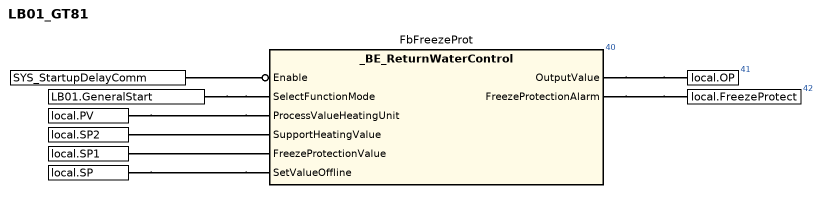
